// TwinCAT 3 PLC project MC
// ProgramVersion: 3.1.4022.2
// libraries:
//   Tc2_MC2, * (Beckhoff Automation GmbH)
//   Tc2_Standard, * (Beckhoff Automation GmbH)
//   Tc2_System, * (Beckhoff Automation GmbH)
//   Tc3_Module, * (Beckhoff Automation GmbH)
// project tree:
//   DUTs/ Command.TcDUT, Status.TcDUT
//   GVLs/ GVL.TcGVL
//   / PlcTask.TcTTO
//   POUs/ BigArm.TcPOU, Clamp.TcPOU, DrivingWheel1.TcPOU, DrivingWheel2.TcPOU, DrivingWheel3.TcPOU, DrivingWheel4.TcPOU, Flex.TcPOU, MAIN.TcPOU, MiddleArm.TcPOU, Rotation.TcPOU, SmallArm.TcPOU, SwingArm1.TcPOU, SwingArm2.TcPOU, SwingArm3.TcPOU, SwingArm4.TcPOU, Waist.TcPOU
// real-time tasks:
//   TASK PlcTask: cycle T#10ms, priority 20, ADS port 350
//   TASK C++task: cycle T#10ms, priority 1, ADS port 351
// motion (NC):
//   TASK NC-Task 1 SAF: cycle T#2ms, priority 4, ADS port 501
//   TASK NC-Task 1 SVB: cycle T#10ms, priority 8, ADS port 511
//   AXIS DrivingWheel1 (id 1)
//     OtherSettings: AllowMotionCmdToSlave=true
//     encoder EncType=19
//       EncPara: ScaleFactorDenominator=29, Inverse=true, MaxCount=#xffffffff
//     drive DrvType=16
//       DrvPara: Inverse=true, MaxCount=#xffffffff
//         Analog: ScaleFactorActTorque=0.1
//         TimeComp: TaskDelayCycles=1
//     controller CtrType=1
//       CtrPara: PriorControlFactor=1
//         Observer: BandWidth=20
//   AXIS DrivingWheel2 (id 2)
//     OtherSettings: AllowMotionCmdToSlave=true
//     encoder EncType=19
//       EncPara: ScaleFactorDenominator=29, Inverse=true, MaxCount=#xffffffff
//     drive DrvType=16
//       DrvPara: Inverse=true, MaxCount=#xffffffff
//         Analog: ScaleFactorActTorque=0.1
//         TimeComp: TaskDelayCycles=1
//     controller CtrType=1
//       CtrPara: PriorControlFactor=1
//         Observer: BandWidth=20
//   AXIS DrivingWheel3 (id 3)
//     OtherSettings: AllowMotionCmdToSlave=true
//     encoder EncType=19
//       EncPara: ScaleFactorDenominator=29, MaxCount=#xffffffff
//     drive DrvType=16
//       DrvPara: MaxCount=#xffffffff
//         Analog: ScaleFactorActTorque=0.1
//         TimeComp: TaskDelayCycles=1
//     controller CtrType=1
//       CtrPara: PriorControlFactor=1
//         Observer: BandWidth=20
//   AXIS DrivingWheel4 (id 4)
//     OtherSettings: AllowMotionCmdToSlave=true
//     encoder EncType=19
//       EncPara: ScaleFactorDenominator=29, MaxCount=#xffffffff
//     drive DrvType=16
//       DrvPara: MaxCount=#xffffffff
//         Analog: ScaleFactorActTorque=0.1
//         TimeComp: TaskDelayCycles=1
//     controller CtrType=1
//       CtrPara: PriorControlFactor=1
//         Observer: BandWidth=20
//   AXIS SwingArm1 (id 5)
//     OtherSettings: AllowMotionCmdToSlave=true
//     encoder EncType=19
//       EncPara: ScaleFactorDenominator=17.3, MaxCount=#xffffffff
//     drive DrvType=16
//       DrvPara: MaxCount=#xffffffff
//         Analog: ScaleFactorActTorque=0.1
//         TimeComp: TaskDelayCycles=1
//     controller CtrType=1
//       CtrPara: PriorControlFactor=1
//         Observer: BandWidth=20
//   AXIS SwingArm2 (id 6)
//     OtherSettings: AllowMotionCmdToSlave=true
//     encoder EncType=19
//       EncPara: ScaleFactorDenominator=17.3, Inverse=true, MaxCount=#xffffffff
//     drive DrvType=16
//       DrvPara: Inverse=true, MaxCount=#xffffffff
//         Analog: ScaleFactorActTorque=0.1
//         TimeComp: TaskDelayCycles=1
//     controller CtrType=1
//       CtrPara: PriorControlFactor=1
//         Observer: BandWidth=20
//   AXIS SwingArm3 (id 7)
//     OtherSettings: AllowMotionCmdToSlave=true
//     encoder EncType=19
//       EncPara: ScaleFactorDenominator=17.3, MaxCount=#xffffffff
//     drive DrvType=16
//       DrvPara: MaxCount=#xffffffff
//         Analog: ScaleFactorActTorque=0.1
//         TimeComp: TaskDelayCycles=1
//     controller CtrType=1
//       CtrPara: PriorControlFactor=1
//         Observer: BandWidth=20
//   AXIS SwingArm4 (id 8)
//     OtherSettings: AllowMotionCmdToSlave=true
//     encoder EncType=19
//       EncPara: ScaleFactorDenominator=17.3, Inverse=true, MaxCount=#xffffffff
//     drive DrvType=16
//       DrvPara: Inverse=true, MaxCount=#xffffffff
//         Analog: ScaleFactorActTorque=0.1
//         TimeComp: TaskDelayCycles=1
//     controller CtrType=1
//       CtrPara: PriorControlFactor=1
//         Observer: BandWidth=20
//   AXIS Waist (id 9)
//     OtherSettings: AllowMotionCmdToSlave=true
//     encoder EncType=19
//       EncPara: MaxCount=#xffffffff
//     drive DrvType=16
//       DrvPara: MaxCount=#xffffffff
//         Analog: ScaleFactorActTorque=0.1
//         TimeComp: TaskDelayCycles=1
//     controller CtrType=1
//       CtrPara: PriorControlFactor=1
//         Observer: BandWidth=20
//   AXIS BigArm (id 10)
//     General: UnitName=Degree
//     Dynamic: AccelerationMaximum=80, DecelerationMaximum=80, Acceleration=80, Deceleration=80, Jerk=80
//     Velo: RefSearch=10, RefSync=10, SlowManual=10, FastManual=55, Maximum=60
//     OtherSettings: AllowMotionCmdToSlave=true, PulseDistancePos=0.5, PulseDistanceNeg=0.5
//     encoder EncType=19
//       EncPara: ScaleFactorNumerator=0.000686645507813, MaxCount=#xffffffff
//     drive DrvType=16
//       DrvPara: MaxCount=#xffffffff
//         Analog: VeloReferenz=60, ScaleFactorActTorque=0.1
//         TimeComp: TaskDelayCycles=1
//     controller CtrType=1
//       CtrPara: PriorControlFactor=1
//         PID: PosKp=7
//         Observer: BandWidth=20
//   AXIS MiddleArm (id 11)
//     General: UnitName=Degree
//     Dynamic: AccelerationMaximum=80, DecelerationMaximum=80, Acceleration=80, Deceleration=80, Jerk=80
//     Velo: RefSearch=10, RefSync=10, SlowManual=10, FastManual=55, Maximum=60
//     OtherSettings: AllowMotionCmdToSlave=true, PulseDistancePos=0.5, PulseDistanceNeg=0.5
//     encoder EncType=19
//       EncPara: ScaleFactorNumerator=0.000686645507813, MaxCount=#xffffffff
//     drive DrvType=16
//       DrvPara: MaxCount=#xffffffff
//         Analog: VeloReferenz=60, ScaleFactorActTorque=0.1
//         TimeComp: TaskDelayCycles=1
//     controller CtrType=1
//       CtrPara: PriorControlFactor=1
//         PID: PosKp=7
//         Observer: BandWidth=20
//   AXIS SmallArm (id 12)
//     General: UnitName=Degree
//     Dynamic: AccelerationMaximum=80, DecelerationMaximum=80, Acceleration=80, Deceleration=80, Jerk=80
//     Velo: RefSearch=10, RefSync=10, SlowManual=10, FastManual=55, Maximum=60
//     OtherSettings: AllowMotionCmdToSlave=true, PulseDistancePos=0.5, PulseDistanceNeg=0.5
//     encoder EncType=19
//       EncPara: ScaleFactorNumerator=0.000686645507813, Inverse=true, MaxCount=#xffffffff
//     drive DrvType=16
//       DrvPara: Inverse=true, MaxCount=#xffffffff
//         Analog: VeloReferenz=60, ScaleFactorActTorque=0.1
//         TimeComp: TaskDelayCycles=1
//     controller CtrType=1
//       CtrPara: PriorControlFactor=1
//         PID: PosKp=7
//         Observer: BandWidth=20
//   AXIS Rotation (id 13)
//     General: UnitName=Degree
//     Dynamic: AccelerationMaximum=80, DecelerationMaximum=80, Acceleration=80, Deceleration=80, Jerk=80
//     Velo: RefSearch=10, RefSync=10, SlowManual=10, FastManual=55, Maximum=60
//     OtherSettings: AllowMotionCmdToSlave=true, PulseDistancePos=0.5, PulseDistanceNeg=0.5
//     encoder EncType=19
//       EncPara: ScaleFactorNumerator=0.000686645507813, MaxCount=#xffffffff
//     drive DrvType=16
//       DrvPara: MaxCount=#xffffffff
//         Analog: VeloReferenz=60, ScaleFactorActTorque=0.1
//         TimeComp: TaskDelayCycles=1
//     controller CtrType=1
//       CtrPara: PriorControlFactor=1
//         PID: PosKp=7
//         Observer: BandWidth=20
// I/O:
//   DEVICE Device 1 (EtherCAT), AmsNetId 192.168.1.200.2.1
//     Term 1 (EK1200) [EK1200-5000 EtherCAT Power supply (2A E-Bus)]
//       Term 2 (EL6751) [EL6751 CANopen Master]
//       Term 3 (EL9011) [EL9011 End Terminal]
//   DEVICE Device 2 (EL6751), AmsNetId 192.168.1.200.3.1
//     Bigarm
//     MiddleArm
//     SmallArm
//     Rotation
//     Box 1 (Twitter)
//   DEVICE Device 5 (EtherCAT), AmsNetId 192.168.1.200.6.1
//     Drive 8 (Elmo Drive) [Gold EtherCAT GCON Drive Rev:0x00010420]
//     Drive 9 (Elmo Drive) [Gold EtherCAT GCON Drive Rev:0x00010420]
//     Drive 10 (Elmo Drive) [Gold EtherCAT GCON Drive Rev:0x00010420]
//     Drive 11 (Elmo Drive) [Gold EtherCAT GCON Drive Rev:0x00010420]
//     Drive 12 (Elmo Drive) [Gold EtherCAT GCON Drive Rev:0x00010420]
//     Drive 13 (Elmo Drive) [Gold EtherCAT GCON Drive Rev:0x00010420]
//     Drive 14 (Elmo Drive) [Gold EtherCAT GCON Drive Rev:0x00010420]
//     Drive 15 (Elmo Drive) [Gold EtherCAT GCON Drive Rev:0x00010420]
//     Drive 16 (Elmo Drive) [Gold EtherCAT GCON Drive Rev:0x00010420]
// variable links:
//   Device 5 (EtherCAT) <-> LibInterface/LibInterface_Obj1 (LibInterface)
//     Drive 11 (Elmo Drive)/Outputs/Digital Outputs <-> Outputs/lighting
//     Drive 15 (Elmo Drive)/Inputs/Digital Inputs <-> Inputs/jinting
//   NC-Task 1 SAF/Axes/BigArm <-> Device 2 (EL6751)/Bigarm
//     Drive/Inputs/In/nState1 <-> TxPDO 3/Inputs/StatusWord1
//     Drive/Inputs/In/nState2 <-> TxPDO 3/Inputs/StatusWord1 @bit 8
//     Drive/Outputs/Out/nCtrl1 <-> RxPDO 3/Outputs/ControlWord1
//     Drive/Outputs/Out/nCtrl2 <-> RxPDO 3/Outputs/ControlWord1 @bit 8
//     Drive/Outputs/Out/nDataOut1 <-> RxPDO 3/Outputs/TargetPosition1
//     Enc/Inputs/In/nDataIn1 <-> TxPDO 3/Inputs/ActualPosition1
//   NC-Task 1 SAF/Axes/DrivingWheel1 <-> Device 5 (EtherCAT)/Drive 8 (Elmo Drive)
//     Drive/Inputs/In/nDcOutputTime <-> InfoData/DcOutputShift
//     Drive/Inputs/In/nState1 <-> Inputs/Status word
//     Drive/Inputs/In/nState2 <-> Inputs/Status word @bit 8
//     Drive/Inputs/In/nState4 @bit 1 <-> WcState/InputToggle
//     Drive/Inputs/In/nState4 <-> WcState/WcState
//     Drive/Outputs/Out/nCtrl1 <-> Outputs/Control word
//     Drive/Outputs/Out/nCtrl2 <-> Outputs/Control word @bit 8
//     Drive/Outputs/Out/nDataOut1 <-> Outputs/Target Position
//     Enc/Inputs/In/nDataIn1 <-> Inputs/Position actual value
//     Enc/Inputs/In/nDcInputTime <-> InfoData/DcInputShift
//     Enc/Inputs/In/nState4 @bit 1 <-> WcState/InputToggle
//     Enc/Inputs/In/nState4 <-> WcState/WcState
//   NC-Task 1 SAF/Axes/DrivingWheel2 <-> Device 5 (EtherCAT)/Drive 10 (Elmo Drive)
//     Drive/Inputs/In/nDcOutputTime <-> InfoData/DcOutputShift
//     Drive/Inputs/In/nState1 <-> Inputs/Status word
//     Drive/Inputs/In/nState2 <-> Inputs/Status word @bit 8
//     Drive/Inputs/In/nState4 @bit 1 <-> WcState/InputToggle
//     Drive/Inputs/In/nState4 <-> WcState/WcState
//     Drive/Outputs/Out/nCtrl1 <-> Outputs/Control word
//     Drive/Outputs/Out/nCtrl2 <-> Outputs/Control word @bit 8
//     Drive/Outputs/Out/nDataOut1 <-> Outputs/Target Position
//     Enc/Inputs/In/nDataIn1 <-> Inputs/Position actual value
//     Enc/Inputs/In/nDcInputTime <-> InfoData/DcInputShift
//     Enc/Inputs/In/nState4 @bit 1 <-> WcState/InputToggle
//     Enc/Inputs/In/nState4 <-> WcState/WcState
//   NC-Task 1 SAF/Axes/DrivingWheel3 <-> Device 5 (EtherCAT)/Drive 12 (Elmo Drive)
//     Drive/Inputs/In/nDcOutputTime <-> InfoData/DcOutputShift
//     Drive/Inputs/In/nState1 <-> Inputs/Status word
//     Drive/Inputs/In/nState2 <-> Inputs/Status word @bit 8
//     Drive/Inputs/In/nState4 @bit 1 <-> WcState/InputToggle
//     Drive/Inputs/In/nState4 <-> WcState/WcState
//     Drive/Outputs/Out/nCtrl1 <-> Outputs/Control word
//     Drive/Outputs/Out/nCtrl2 <-> Outputs/Control word @bit 8
//     Drive/Outputs/Out/nDataOut1 <-> Outputs/Target Position
//     Enc/Inputs/In/nDataIn1 <-> Inputs/Position actual value
//     Enc/Inputs/In/nDcInputTime <-> InfoData/DcInputShift
//     Enc/Inputs/In/nState4 @bit 1 <-> WcState/InputToggle
//     Enc/Inputs/In/nState4 <-> WcState/WcState
//   NC-Task 1 SAF/Axes/DrivingWheel4 <-> Device 5 (EtherCAT)/Drive 14 (Elmo Drive)
//     Drive/Inputs/In/nDcOutputTime <-> InfoData/DcOutputShift
//     Drive/Inputs/In/nState1 <-> Inputs/Status word
//     Drive/Inputs/In/nState2 <-> Inputs/Status word @bit 8
//     Drive/Inputs/In/nState4 @bit 1 <-> WcState/InputToggle
//     Drive/Inputs/In/nState4 <-> WcState/WcState
//     Drive/Outputs/Out/nCtrl1 <-> Outputs/Control word
//     Drive/Outputs/Out/nCtrl2 <-> Outputs/Control word @bit 8
//     Drive/Outputs/Out/nDataOut1 <-> Outputs/Target Position
//     Enc/Inputs/In/nDataIn1 <-> Inputs/Position actual value
//     Enc/Inputs/In/nDcInputTime <-> InfoData/DcInputShift
//     Enc/Inputs/In/nState4 @bit 1 <-> WcState/InputToggle
//     Enc/Inputs/In/nState4 <-> WcState/WcState
//   NC-Task 1 SAF/Axes/MiddleArm <-> Device 2 (EL6751)/MiddleArm
//     Drive/Inputs/In/nState1 <-> TxPDO 3/Inputs/StatusWord1
//     Drive/Inputs/In/nState2 <-> TxPDO 3/Inputs/StatusWord1 @bit 8
//     Drive/Outputs/Out/nCtrl1 <-> RxPDO 3/Outputs/ControlWord1
//     Drive/Outputs/Out/nCtrl2 <-> RxPDO 3/Outputs/ControlWord1 @bit 8
//     Drive/Outputs/Out/nDataOut1 <-> RxPDO 3/Outputs/TargetPosition1
//     Enc/Inputs/In/nDataIn1 <-> TxPDO 3/Inputs/ActualPosition1
//   NC-Task 1 SAF/Axes/Rotation <-> Device 2 (EL6751)/Rotation
//     Drive/Inputs/In/nState1 <-> TxPDO 3/Inputs/StatusWord1
//     Drive/Inputs/In/nState2 <-> TxPDO 3/Inputs/StatusWord1 @bit 8
//     Drive/Outputs/Out/nCtrl1 <-> RxPDO 3/Outputs/ControlWord1
//     Drive/Outputs/Out/nCtrl2 <-> RxPDO 3/Outputs/ControlWord1 @bit 8
//     Drive/Outputs/Out/nDataOut1 <-> RxPDO 3/Outputs/TargetPosition1
//     Enc/Inputs/In/nDataIn1 <-> TxPDO 3/Inputs/ActualPosition1
//   NC-Task 1 SAF/Axes/SmallArm <-> Device 2 (EL6751)/SmallArm
//     Drive/Inputs/In/nState1 <-> TxPDO 3/Inputs/StatusWord1
//     Drive/Inputs/In/nState2 <-> TxPDO 3/Inputs/StatusWord1 @bit 8
//     Drive/Outputs/Out/nCtrl1 <-> RxPDO 3/Outputs/ControlWord1
//     Drive/Outputs/Out/nCtrl2 <-> RxPDO 3/Outputs/ControlWord1 @bit 8
//     Drive/Outputs/Out/nDataOut1 <-> RxPDO 3/Outputs/TargetPosition1
//     Enc/Inputs/In/nDataIn1 <-> TxPDO 3/Inputs/ActualPosition1
//   NC-Task 1 SAF/Axes/SwingArm1 <-> Device 5 (EtherCAT)/Drive 9 (Elmo Drive)
//     Drive/Inputs/In/nDcOutputTime <-> InfoData/DcOutputShift
//     Drive/Inputs/In/nState1 <-> Inputs/Status word
//     Drive/Inputs/In/nState2 <-> Inputs/Status word @bit 8
//     Drive/Inputs/In/nState4 @bit 1 <-> WcState/InputToggle
//     Drive/Inputs/In/nState4 <-> WcState/WcState
//     Drive/Outputs/Out/nCtrl1 <-> Outputs/Control word
//     Drive/Outputs/Out/nCtrl2 <-> Outputs/Control word @bit 8
//     Drive/Outputs/Out/nDataOut1 <-> Outputs/Target Position
//     Enc/Inputs/In/nDataIn1 <-> Inputs/Position actual value
//     Enc/Inputs/In/nDcInputTime <-> InfoData/DcInputShift
//     Enc/Inputs/In/nState4 @bit 1 <-> WcState/InputToggle
//     Enc/Inputs/In/nState4 <-> WcState/WcState
//   NC-Task 1 SAF/Axes/SwingArm2 <-> Device 5 (EtherCAT)/Drive 11 (Elmo Drive)
//     Drive/Inputs/In/nDcOutputTime <-> InfoData/DcOutputShift
//     Drive/Inputs/In/nState1 <-> Inputs/Status word
//     Drive/Inputs/In/nState2 <-> Inputs/Status word @bit 8
//     Drive/Inputs/In/nState4 @bit 1 <-> WcState/InputToggle
//     Drive/Inputs/In/nState4 <-> WcState/WcState
//     Drive/Outputs/Out/nCtrl1 <-> Outputs/Control word
//     Drive/Outputs/Out/nCtrl2 <-> Outputs/Control word @bit 8
//     Drive/Outputs/Out/nDataOut1 <-> Outputs/Target Position
//     Enc/Inputs/In/nDataIn1 <-> Inputs/Position actual value
//     Enc/Inputs/In/nDcInputTime <-> InfoData/DcInputShift
//     Enc/Inputs/In/nState4 @bit 1 <-> WcState/InputToggle
//     Enc/Inputs/In/nState4 <-> WcState/WcState
//   NC-Task 1 SAF/Axes/SwingArm3 <-> Device 5 (EtherCAT)/Drive 13 (Elmo Drive)
//     Drive/Inputs/In/nDcOutputTime <-> InfoData/DcOutputShift
//     Drive/Inputs/In/nState1 <-> Inputs/Status word
//     Drive/Inputs/In/nState2 <-> Inputs/Status word @bit 8
//     Drive/Inputs/In/nState4 @bit 1 <-> WcState/InputToggle
//     Drive/Inputs/In/nState4 <-> WcState/WcState
//     Drive/Outputs/Out/nCtrl1 <-> Outputs/Control word
//     Drive/Outputs/Out/nCtrl2 <-> Outputs/Control word @bit 8
//     Drive/Outputs/Out/nDataOut1 <-> Outputs/Target Position
//     Enc/Inputs/In/nDataIn1 <-> Inputs/Position actual value
//     Enc/Inputs/In/nDcInputTime <-> InfoData/DcInputShift
//     Enc/Inputs/In/nState4 @bit 1 <-> WcState/InputToggle
//     Enc/Inputs/In/nState4 <-> WcState/WcState
//   NC-Task 1 SAF/Axes/SwingArm4 <-> Device 5 (EtherCAT)/Drive 15 (Elmo Drive)
//     Drive/Inputs/In/nDcOutputTime <-> InfoData/DcOutputShift
//     Drive/Inputs/In/nState1 <-> Inputs/Status word
//     Drive/Inputs/In/nState2 <-> Inputs/Status word @bit 8
//     Drive/Inputs/In/nState4 @bit 1 <-> WcState/InputToggle
//     Drive/Inputs/In/nState4 <-> WcState/WcState
//     Drive/Outputs/Out/nCtrl1 <-> Outputs/Control word
//     Drive/Outputs/Out/nCtrl2 <-> Outputs/Control word @bit 8
//     Drive/Outputs/Out/nDataOut1 <-> Outputs/Target Position
//     Enc/Inputs/In/nDataIn1 <-> Inputs/Position actual value
//     Enc/Inputs/In/nDcInputTime <-> InfoData/DcInputShift
//     Enc/Inputs/In/nState4 @bit 1 <-> WcState/InputToggle
//     Enc/Inputs/In/nState4 <-> WcState/WcState
//   NC-Task 1 SAF/Axes/Waist <-> Device 5 (EtherCAT)/Drive 16 (Elmo Drive)
//     Drive/Inputs/In/nDcOutputTime <-> InfoData/DcOutputShift
//     Drive/Inputs/In/nState1 <-> Inputs/Status word
//     Drive/Inputs/In/nState2 <-> Inputs/Status word @bit 8
//     Drive/Inputs/In/nState4 @bit 1 <-> WcState/InputToggle
//     Drive/Inputs/In/nState4 <-> WcState/WcState
//     Drive/Outputs/Out/nCtrl1 <-> Outputs/Control word
//     Drive/Outputs/Out/nCtrl2 <-> Outputs/Control word @bit 8
//     Drive/Outputs/Out/nDataOut1 <-> Outputs/Target Position
//     Enc/Inputs/In/nDataIn1 <-> Inputs/Position actual value
//     Enc/Inputs/In/nDcInputTime <-> InfoData/DcInputShift
//     Enc/Inputs/In/nState4 @bit 1 <-> WcState/InputToggle
//     Enc/Inputs/In/nState4 <-> WcState/WcState
//   MC/MC Instance <-> Device 2 (EL6751)/Box 1 (Twitter)
//     PlcTask Inputs/GVL.Astatusword[1] <-> TxPDO 1/Inputs/statusword
//     PlcTask Inputs/GVL.readActualpostion[1] <-> TxPDO 1/Inputs/Actualpostion
//     PlcTask Inputs/GVL.readIOStatus[1] <-> TxPDO 2/Inputs/DI
//     PlcTask Outputs/GVL.Acontrolword[1] <-> RxPDO 1/Outputs/Controlword
//     PlcTask Outputs/GVL.SetActualVelocity[1] <-> RxPDO 2/Outputs/TargetVelocity
//     PlcTask Outputs/GVL.SetUnitmode[1] <-> RxPDO 2/Outputs/unitmode
//   MC/MC Instance <-> NC-Task 1 SAF/Axes/BigArm
//     PlcTask Inputs/MAIN.fbBigArm.axis.NcToPlc <-> Outputs/ToPlc
//     PlcTask Outputs/MAIN.fbBigArm.axis.PlcToNc <-> Inputs/FromPlc
//   MC/MC Instance <-> NC-Task 1 SAF/Axes/DrivingWheel1
//     PlcTask Inputs/MAIN.fbDrivingWheel1.axis.NcToPlc <-> Outputs/ToPlc
//     PlcTask Outputs/MAIN.fbDrivingWheel1.axis.PlcToNc <-> Inputs/FromPlc
//   MC/MC Instance <-> NC-Task 1 SAF/Axes/DrivingWheel2
//     PlcTask Inputs/MAIN.fbDrivingWheel2.axis.NcToPlc <-> Outputs/ToPlc
//     PlcTask Outputs/MAIN.fbDrivingWheel2.axis.PlcToNc <-> Inputs/FromPlc
//   MC/MC Instance <-> NC-Task 1 SAF/Axes/DrivingWheel3
//     PlcTask Inputs/MAIN.fbDrivingWheel3.axis.NcToPlc <-> Outputs/ToPlc
//     PlcTask Outputs/MAIN.fbDrivingWheel3.axis.PlcToNc <-> Inputs/FromPlc
//   MC/MC Instance <-> NC-Task 1 SAF/Axes/DrivingWheel4
//     PlcTask Inputs/MAIN.fbDrivingWheel4.axis.NcToPlc <-> Outputs/ToPlc
//     PlcTask Outputs/MAIN.fbDrivingWheel4.axis.PlcToNc <-> Inputs/FromPlc
//   MC/MC Instance <-> NC-Task 1 SAF/Axes/MiddleArm
//     PlcTask Inputs/MAIN.fbMiddleArm.axis.NcToPlc <-> Outputs/ToPlc
//     PlcTask Outputs/MAIN.fbMiddleArm.axis.PlcToNc <-> Inputs/FromPlc
//   MC/MC Instance <-> NC-Task 1 SAF/Axes/Rotation
//     PlcTask Inputs/MAIN.fbRotation.axis.NcToPlc <-> Outputs/ToPlc
//     PlcTask Outputs/MAIN.fbRotation.axis.PlcToNc <-> Inputs/FromPlc
//   MC/MC Instance <-> NC-Task 1 SAF/Axes/SmallArm
//     PlcTask Inputs/MAIN.fbSmallArm.axis.NcToPlc <-> Outputs/ToPlc
//     PlcTask Outputs/MAIN.fbSmallArm.axis.PlcToNc <-> Inputs/FromPlc
//   MC/MC Instance <-> NC-Task 1 SAF/Axes/SwingArm1
//     PlcTask Inputs/MAIN.fbSwingArm1.axis.NcToPlc <-> Outputs/ToPlc
//     PlcTask Outputs/MAIN.fbSwingArm1.axis.PlcToNc <-> Inputs/FromPlc
//   MC/MC Instance <-> NC-Task 1 SAF/Axes/SwingArm2
//     PlcTask Inputs/MAIN.fbSwingArm2.axis.NcToPlc <-> Outputs/ToPlc
//     PlcTask Outputs/MAIN.fbSwingArm2.axis.PlcToNc <-> Inputs/FromPlc
//   MC/MC Instance <-> NC-Task 1 SAF/Axes/SwingArm3
//     PlcTask Inputs/MAIN.fbSwingArm3.axis.NcToPlc <-> Outputs/ToPlc
//     PlcTask Outputs/MAIN.fbSwingArm3.axis.PlcToNc <-> Inputs/FromPlc
//   MC/MC Instance <-> NC-Task 1 SAF/Axes/SwingArm4
//     PlcTask Inputs/MAIN.fbSwingArm4.axis.NcToPlc <-> Outputs/ToPlc
//     PlcTask Outputs/MAIN.fbSwingArm4.axis.PlcToNc <-> Inputs/FromPlc
//   MC/MC Instance <-> NC-Task 1 SAF/Axes/Waist
//     PlcTask Inputs/MAIN.fbWaist.axis.NcToPlc <-> Outputs/ToPlc
//     PlcTask Outputs/MAIN.fbWaist.axis.PlcToNc <-> Inputs/FromPlc
//   MC/MC Instance <-> LibInterface/LibInterface_Obj1 (LibInterface)
//     PlcTask Inputs/MAIN.BigArmInput/Enable <-> Outputs/BigArmInput/Enable
//     PlcTask Inputs/MAIN.BigArmInput/Halt <-> Outputs/BigArmInput/Halt
//     PlcTask Inputs/MAIN.BigArmInput/Home <-> Outputs/BigArmInput/Home
//     PlcTask Inputs/MAIN.BigArmInput/Move_Absolute <-> Outputs/BigArmInput/MoveAbsolute
//     PlcTask Inputs/MAIN.BigArmInput/Move_Relative <-> Outputs/BigArmInput/MoveRelative
//     PlcTask Inputs/MAIN.BigArmInput/Move_Velocity <-> Outputs/BigArmInput/MoveVelocity
//     PlcTask Inputs/MAIN.BigArmInput/Position <-> Outputs/BigArmInput/Position
//     PlcTask Inputs/MAIN.BigArmInput/Reset <-> Outputs/BigArmInput/Reset
//     PlcTask Inputs/MAIN.BigArmInput/SetZero <-> Outputs/BigArmInput/SetZero
//     PlcTask Inputs/MAIN.BigArmInput/Velocity <-> Outputs/BigArmInput/Velocity
//     PlcTask Inputs/MAIN.DrivingWheel{1..4}Input/Enable <-> Outputs/DrivingWheel{1..4}Input/Enable  (4 links)
//     PlcTask Inputs/MAIN.DrivingWheel{1..4}Input/Halt <-> Outputs/DrivingWheel{1..4}Input/Halt  (4 links)
//     PlcTask Inputs/MAIN.DrivingWheel{1..4}Input/Home <-> Outputs/DrivingWheel{1..4}Input/Home  (4 links)
//     PlcTask Inputs/MAIN.DrivingWheel{1..4}Input/Move_Absolute <-> Outputs/DrivingWheel{1..4}Input/MoveAbsolute  (4 links)
//     PlcTask Inputs/MAIN.DrivingWheel{1..4}Input/Move_Relative <-> Outputs/DrivingWheel{1..4}Input/MoveRelative  (4 links)
//     PlcTask Inputs/MAIN.DrivingWheel{1..4}Input/Move_Velocity <-> Outputs/DrivingWheel{1..4}Input/MoveVelocity  (4 links)
//     PlcTask Inputs/MAIN.DrivingWheel{1..4}Input/Position <-> Outputs/DrivingWheel{1..4}Input/Position  (4 links)
//     PlcTask Inputs/MAIN.DrivingWheel{1..4}Input/Reset <-> Outputs/DrivingWheel{1..4}Input/Reset  (4 links)
//     PlcTask Inputs/MAIN.DrivingWheel{1..4}Input/SetZero <-> Outputs/DrivingWheel{1..4}Input/SetZero  (4 links)
//     PlcTask Inputs/MAIN.DrivingWheel{1..4}Input/Velocity <-> Outputs/DrivingWheel{1..4}Input/Velocity  (4 links)
//     PlcTask Inputs/MAIN.FlexInput/Enable <-> Outputs/FlexInput/Enable
//     PlcTask Inputs/MAIN.FlexInput/Halt <-> Outputs/FlexInput/Halt
//     PlcTask Inputs/MAIN.FlexInput/Home <-> Outputs/FlexInput/Home
//     PlcTask Inputs/MAIN.FlexInput/Move_Absolute <-> Outputs/FlexInput/MoveAbsolute
//     PlcTask Inputs/MAIN.FlexInput/Move_Relative <-> Outputs/FlexInput/MoveRelative
//     PlcTask Inputs/MAIN.FlexInput/Move_Velocity <-> Outputs/FlexInput/MoveVelocity
//     PlcTask Inputs/MAIN.FlexInput/Position <-> Outputs/FlexInput/Position
//     PlcTask Inputs/MAIN.FlexInput/Reset <-> Outputs/FlexInput/Reset
//     PlcTask Inputs/MAIN.FlexInput/SetZero <-> Outputs/FlexInput/SetZero
//     PlcTask Inputs/MAIN.FlexInput/Velocity <-> Outputs/FlexInput/Velocity
//     PlcTask Inputs/MAIN.GripperEnable <-> Outputs/ClampInput/Enable
//     PlcTask Inputs/MAIN.GripperSetSpeed <-> Outputs/ClampInput/SetSpped
//     PlcTask Inputs/MAIN.MiddleArmInput/Enable <-> Outputs/MiddleArmInput/Enable
//     PlcTask Inputs/MAIN.MiddleArmInput/Halt <-> Outputs/MiddleArmInput/Halt
//     PlcTask Inputs/MAIN.MiddleArmInput/Home <-> Outputs/MiddleArmInput/Home
//     PlcTask Inputs/MAIN.MiddleArmInput/Move_Absolute <-> Outputs/MiddleArmInput/MoveAbsolute
//     PlcTask Inputs/MAIN.MiddleArmInput/Move_Relative <-> Outputs/MiddleArmInput/MoveRelative
//     PlcTask Inputs/MAIN.MiddleArmInput/Move_Velocity <-> Outputs/MiddleArmInput/MoveVelocity
//     PlcTask Inputs/MAIN.MiddleArmInput/Position <-> Outputs/MiddleArmInput/Position
//     PlcTask Inputs/MAIN.MiddleArmInput/Reset <-> Outputs/MiddleArmInput/Reset
//     PlcTask Inputs/MAIN.MiddleArmInput/SetZero <-> Outputs/MiddleArmInput/SetZero
//     PlcTask Inputs/MAIN.MiddleArmInput/Velocity <-> Outputs/MiddleArmInput/Velocity
//     PlcTask Inputs/MAIN.RotationInput/Enable <-> Outputs/RotationInput/Enable
//     PlcTask Inputs/MAIN.RotationInput/Halt <-> Outputs/RotationInput/Halt
//     PlcTask Inputs/MAIN.RotationInput/Home <-> Outputs/RotationInput/Home
//     PlcTask Inputs/MAIN.RotationInput/Move_Absolute <-> Outputs/RotationInput/MoveAbsolute
//     PlcTask Inputs/MAIN.RotationInput/Move_Relative <-> Outputs/RotationInput/MoveRelative
//     PlcTask Inputs/MAIN.RotationInput/Move_Velocity <-> Outputs/RotationInput/MoveVelocity
//     PlcTask Inputs/MAIN.RotationInput/Position <-> Outputs/RotationInput/Position
//     PlcTask Inputs/MAIN.RotationInput/Reset <-> Outputs/RotationInput/Reset
//     PlcTask Inputs/MAIN.RotationInput/SetZero <-> Outputs/RotationInput/SetZero
//     PlcTask Inputs/MAIN.RotationInput/Velocity <-> Outputs/RotationInput/Velocity
//     PlcTask Inputs/MAIN.SmallArmInput/Enable <-> Outputs/SmallArmInput/Enable
//     PlcTask Inputs/MAIN.SmallArmInput/Halt <-> Outputs/SmallArmInput/Halt
//     PlcTask Inputs/MAIN.SmallArmInput/Home <-> Outputs/SmallArmInput/Home
//     PlcTask Inputs/MAIN.SmallArmInput/Move_Absolute <-> Outputs/SmallArmInput/MoveAbsolute
//     PlcTask Inputs/MAIN.SmallArmInput/Move_Relative <-> Outputs/SmallArmInput/MoveRelative
//     PlcTask Inputs/MAIN.SmallArmInput/Move_Velocity <-> Outputs/SmallArmInput/MoveVelocity
//     PlcTask Inputs/MAIN.SmallArmInput/Position <-> Outputs/SmallArmInput/Position
//     PlcTask Inputs/MAIN.SmallArmInput/Reset <-> Outputs/SmallArmInput/Reset
//     PlcTask Inputs/MAIN.SmallArmInput/SetZero <-> Outputs/SmallArmInput/SetZero
//     PlcTask Inputs/MAIN.SmallArmInput/Velocity <-> Outputs/SmallArmInput/Velocity
//     PlcTask Inputs/MAIN.SwingArm{1..4}Input/Enable <-> Outputs/SwingArm{1..4}Input/Enable  (4 links)
//     PlcTask Inputs/MAIN.SwingArm{1..4}Input/Halt <-> Outputs/SwingArm{1..4}Input/Halt  (4 links)
//     PlcTask Inputs/MAIN.SwingArm{1..4}Input/Home <-> Outputs/SwingArm{1..4}Input/Home  (4 links)
//     PlcTask Inputs/MAIN.SwingArm{1..4}Input/Move_Absolute <-> Outputs/SwingArm{1..4}Input/MoveAbsolute  (4 links)
//     PlcTask Inputs/MAIN.SwingArm{1..4}Input/Move_Relative <-> Outputs/SwingArm{1..4}Input/MoveRelative  (4 links)
//     PlcTask Inputs/MAIN.SwingArm{1..4}Input/Move_Velocity <-> Outputs/SwingArm{1..4}Input/MoveVelocity  (4 links)
//     PlcTask Inputs/MAIN.SwingArm{1..4}Input/Position <-> Outputs/SwingArm{1..4}Input/Position  (4 links)
//     PlcTask Inputs/MAIN.SwingArm{1..4}Input/Reset <-> Outputs/SwingArm{1..4}Input/Reset  (4 links)
//     PlcTask Inputs/MAIN.SwingArm{1..4}Input/SetZero <-> Outputs/SwingArm{1..4}Input/SetZero  (4 links)
//     PlcTask Inputs/MAIN.SwingArm{1..4}Input/Velocity <-> Outputs/SwingArm{1..4}Input/Velocity  (4 links)
//     PlcTask Inputs/MAIN.WaistInput/Enable <-> Outputs/WaistInput/Enable
//     PlcTask Inputs/MAIN.WaistInput/Halt <-> Outputs/WaistInput/Halt
//     PlcTask Inputs/MAIN.WaistInput/Home <-> Outputs/WaistInput/Home
//     PlcTask Inputs/MAIN.WaistInput/Move_Absolute <-> Outputs/WaistInput/MoveAbsolute
//     PlcTask Inputs/MAIN.WaistInput/Move_Relative <-> Outputs/WaistInput/MoveRelative
//     PlcTask Inputs/MAIN.WaistInput/Move_Velocity <-> Outputs/WaistInput/MoveVelocity
//     PlcTask Inputs/MAIN.WaistInput/Position <-> Outputs/WaistInput/Position
//     PlcTask Inputs/MAIN.WaistInput/Reset <-> Outputs/WaistInput/Reset
//     PlcTask Inputs/MAIN.WaistInput/SetZero <-> Outputs/WaistInput/SetZero
//     PlcTask Inputs/MAIN.WaistInput/Velocity <-> Outputs/WaistInput/Velocity
//     PlcTask Outputs/MAIN.BigArmOutput/Enable <-> Inputs/BigArmOutput/Enable
//     PlcTask Outputs/MAIN.BigArmOutput/Position <-> Inputs/BigArmOutput/Position
//     PlcTask Outputs/MAIN.BigArmOutput/Velocity <-> Inputs/BigArmOutput/Velocity
//     PlcTask Outputs/MAIN.DrivingWheel{1..4}Output/Enable <-> Inputs/DrivingWheel{1..4}Output/Enable  (4 links)
//     PlcTask Outputs/MAIN.DrivingWheel{1..4}Output/Position <-> Inputs/DrivingWheel{1..4}Output/Position  (4 links)
//     PlcTask Outputs/MAIN.DrivingWheel{1..4}Output/Velocity <-> Inputs/DrivingWheel{1..4}Output/Velocity  (4 links)
//     PlcTask Outputs/MAIN.FlexOutput/Enable <-> Inputs/FlexOutput/Enable
//     PlcTask Outputs/MAIN.FlexOutput/Position <-> Inputs/FlexOutput/Position
//     PlcTask Outputs/MAIN.FlexOutput/Velocity <-> Inputs/FlexOutput/Velocity
//     PlcTask Outputs/MAIN.GripperIOStatus <-> Inputs/ClampOutput/IO
//     PlcTask Outputs/MAIN.GripperReadPos <-> Inputs/ClampOutput/Position
//     PlcTask Outputs/MAIN.MiddleArmOutput/Enable <-> Inputs/MiddleArmOutput/Enable
//     PlcTask Outputs/MAIN.MiddleArmOutput/Position <-> Inputs/MiddleArmOutput/Position
//     PlcTask Outputs/MAIN.MiddleArmOutput/Velocity <-> Inputs/MiddleArmOutput/Velocity
//     PlcTask Outputs/MAIN.RotationOutput/Enable <-> Inputs/RotationOutput/Enable
//     PlcTask Outputs/MAIN.RotationOutput/Position <-> Inputs/RotationOutput/Position
//     PlcTask Outputs/MAIN.RotationOutput/Velocity <-> Inputs/RotationOutput/Velocity
//     PlcTask Outputs/MAIN.SmallArmOutput/Enable <-> Inputs/SmallArmOutput/Enable
//     PlcTask Outputs/MAIN.SmallArmOutput/Position <-> Inputs/SmallArmOutput/Position
//     PlcTask Outputs/MAIN.SmallArmOutput/Velocity <-> Inputs/SmallArmOutput/Velocity
//     PlcTask Outputs/MAIN.SwingArm{1..4}Output/Enable <-> Inputs/SwingArm{1..4}Output/Enable  (4 links)
//     PlcTask Outputs/MAIN.SwingArm{1..4}Output/Position <-> Inputs/SwingArm{1..4}Output/Position  (4 links)
//     PlcTask Outputs/MAIN.SwingArm{1..4}Output/Velocity <-> Inputs/SwingArm{1..4}Output/Velocity  (4 links)
//     PlcTask Outputs/MAIN.WaistOutput/Enable <-> Inputs/WaistOutput/Enable
//     PlcTask Outputs/MAIN.WaistOutput/Position <-> Inputs/WaistOutput/Position
//     PlcTask Outputs/MAIN.WaistOutput/Velocity <-> Inputs/WaistOutput/Velocity

CONFIGURATION MC
    RESOURCE PLC ON TwinCAT3
        TASK PlcTask(INTERVAL := T#10ms, PRIORITY := 20);
        PROGRAM MAIN WITH PlcTask : MAIN;
    END_RESOURCE
END_CONFIGURATION

// ---- DUTs/Command.TcDUT
TYPE Command :
STRUCT
	Enable:BOOL;					//使能触发位
	Move_Absolute:BOOL;				//绝对运动触发位
	Move_Relative:BOOL;				//相对运动触发位
	Move_Velocity:BOOL;				//匀速运动触发位
	Reset:BOOL;						//复位触发位
	Halt:BOOL;						//暂停触发位
	Home:BOOL;						//暂停触发位
	SetZero:BOOL;					//设置位置触发位
	Velocity:LREAL;					//速度变量
	Position:LREAL;					//位置变量
	HomeSignal:DINT;				//寻参触发点
END_STRUCT
END_TYPE

// ---- DUTs/Status.TcDUT
TYPE Status :
STRUCT
	Enable:BOOL;					//使能状态
	Velocity:LREAL;					//速度状态
	Position:LREAL;					//位置状态
END_STRUCT
END_TYPE

// ---- GVLs/GVL.TcGVL
{attribute 'qualified_only'}
VAR_GLOBAL
	Acontrolword  AT%Q*:ARRAY[1..1]OF UINT;
	
	SetActualVelocity AT%Q*:ARRAY[1..1]OF DINT;
	SetUnitmode AT%Q*:ARRAY[1..1]OF BYTE;
	
	
	
	Astatusword AT%I*:ARRAY[1..1]OF UINT;
	readActualpostion AT%I*:ARRAY[1..1]OF DINT;
	readActualCurrent AT%I*:ARRAY[1..1]OF UINT;
	readIOStatus AT%I*:ARRAY[1..1]OF DINT;
	
	bigarm_position:LREAL;
	middlearm_position:LREAL;
	
	
	
END_VAR

// ---- POUs/MAIN.TcPOU
PROGRAM MAIN
VAR
	fbDrivingWheel1:DrivingWheel1;				//调用控制驱动轮1功能块
	fbDrivingWheel2:DrivingWheel2;				//调用控制驱动轮2功能块
	fbDrivingWheel3:DrivingWheel3;				//调用控制驱动轮3功能块
	fbDrivingWheel4:DrivingWheel4;				//调用控制驱动轮4功能块
	fbSwingArm1:SwingArm1;						//调用控制摆臂1功能块
	fbSwingArm2:SwingArm2;						//调用控制摆臂2功能块
	fbSwingArm3:SwingArm3;						//调用控制摆臂3功能块
	fbSwingArm4:SwingArm4;						//调用控制摆臂4功能块
	fbWaist:Waist;								//调用控制腰功能块
	fbBigArm:BigArm;							//调用控制大臂功能块
	fbFlex:Flex;								//调用控制伸缩功能块
	fbMiddleArm:MiddleArm;						//调用控制中臂功能块
	fbSmallArm:SmallArm;						//调用控制小臂功能块
	fbRotation:Rotation;						//调用控制旋转功能块
	fbClamp:Clamp;								//调用控制夹紧功能块
//***************************************************************//
	DrivingWheel1Input AT%I*:Command;//驱动轮1PLC轴输入变量
	DrivingWheel2Input AT%I*:Command;//驱动轮2PLC轴输入变量
	DrivingWheel3Input AT%I*:Command;//驱动轮3PLC轴输入变量
	DrivingWheel4Input AT%I*:Command;//驱动轮4PLC轴输入变量
	SwingArm1Input AT%I*:Command;	 //摆臂1PLC轴输入变量
	SwingArm2Input AT%I*:Command;	 //摆臂2PLC轴输入变量
	SwingArm3Input AT%I*:Command;	 //摆臂3PLC轴输入变量
	SwingArm4Input AT%I*:Command;	 //摆臂4PLC轴输入变量
	WaistInput AT%I*:Command;	 	 //腰PLC轴输入变量
	BigArmInput AT%I*:Command;		 //大臂PLC轴输入变量
	FlexInput AT%I*:Command;		 //伸缩PLC轴输入变量
	MiddleArmInput AT%I*:Command;	 //中臂PLC轴输入变量
	SmallArmInput AT%I*:Command;	 //小臂PLC轴输入变量
	RotationInput AT%I*:Command;	 //旋转PLC轴输入变量
	ClampInput AT%I*:Command;		 //夹紧PLC轴输入变量
//***************************************************************//
	DrivingWheel1Output AT%Q*:Status;//驱动轮1PLC轴输出变量
	DrivingWheel2Output AT%Q*:Status;//驱动轮2PLC轴输出变量
	DrivingWheel3Output AT%Q*:Status;//驱动轮3LC轴输出变量
	DrivingWheel4Output AT%Q*:Status;//驱动轮4PLC轴输出变量
	SwingArm1Output AT%Q*:Status;//摆臂1PLC轴输出变量
	SwingArm2Output AT%Q*:Status;//摆臂2PLC轴输出变量
	SwingArm3Output AT%Q*:Status;//摆臂3PLC轴输出变量
	SwingArm4Output AT%Q*:Status;//摆臂4PLC轴输出变量
	WaistOutput AT%Q*:Status; //腰PLC轴输出变量
	BigArmOutput AT%Q*:Status;//大臂PLC轴输出变量
	FlexOutput AT%Q*:Status; //伸缩PLC轴输出变量
	MiddleArmOutput AT%Q*:Status;//中臂PLC轴输出变量
	SmallArmOutput AT%Q*:Status;//小臂PLC轴输出变量
	RotationOutput AT%Q*:Status;//旋转PLC轴输出变量
	ClampOutput AT%Q*:Status;//夹紧PLC轴输出变量
	///////////////////////////////////////////////////////
	GripperEnable AT%I*:DINT;
	GripperSetSpeed AT%I*:DINT;
	GripperReadPos AT%Q*:DINT;
	GripperIOStatus AT%Q*:DINT;
END_VAR


fbDrivingWheel1( AxisInput:=DrivingWheel1Input , AxisOutput=>DrivingWheel1Output );
fbDrivingWheel2( AxisInput:=DrivingWheel2Input , AxisOutput=>DrivingWheel2Output );
fbDrivingWheel3( AxisInput:=DrivingWheel3Input , AxisOutput=>DrivingWheel3Output );
fbDrivingWheel4( AxisInput:=DrivingWheel4Input , AxisOutput=>DrivingWheel4Output );

fbSwingArm1( AxisInput:=SwingArm1Input , AxisOutput=>SwingArm1Output );
fbSwingArm2( AxisInput:=SwingArm2Input , AxisOutput=>SwingArm2Output );
fbSwingArm3( AxisInput:=SwingArm3Input , AxisOutput=>SwingArm3Output );
fbSwingArm4( AxisInput:=SwingArm4Input , AxisOutput=>SwingArm4Output );

fbWaist( AxisInput:=WaistInput , AxisOutput=>WaistOutput );
fbBigArm( AxisInput:=BigArmInput , AxisOutput=>BigArmOutput );
fbFlex(AxisInput:=FlexInput, AxisOutput=>FlexOutput);
fbMiddleArm( AxisInput:=MiddleArmInput , AxisOutput=>MiddleArmOutput );
fbSmallArm( AxisInput:=SmallArmInput , AxisOutput=>SmallArmOutput );
fbRotation( AxisInput:=RotationInput , AxisOutput=>RotationOutput );
fbClamp( AxisInput:=ClampInput , AxisOutput=>ClampOutput );

//////////////////////////////////////////////////////////////////////
//Enable
//when receive enable signal,then gripper driver would be enabled in 3 circles
IF(GripperEnable=1 AND NOT(GVL.Acontrolword[1] =15))THEN
	IF(NOT(GVL.Acontrolword[1] =6) AND NOT(GVL.Acontrolword[1] =7))THEN
			GVL.Acontrolword[1] :=6;		
	ELSIF(GVL.Acontrolword[1] =6)THEN
			GVL.Acontrolword[1] :=7;	
	ELSE
			GVL.Acontrolword[1] :=15;	
			//set driver mode
			GVL.SetUnitmode[1]:=3;
	END_IF
END_IF

//disable
//when receive disnable signal,then gripper driver would be disnabled immediately
IF(GripperEnable=0)THEN
	GVL.Acontrolword[1] :=0;	
END_IF


//set gripper speed,positive speed represent open ,negative speed represent close
IF(GripperEnable=1)THEN
	IF(GripperSetSpeed>100)THEN
		GVL.SetActualVelocity[1]:=100*1000;
	ELSIF(GripperSetSpeed<-100)THEN
		GVL.SetActualVelocity[1]:=-100*1000;
	END_IF
	GVL.SetActualVelocity[1]:=GripperSetSpeed*1000;
END_IF
GripperReadPos:=GVL.readActualpostion[1];
//18bit is the postion-constraint switch
GripperIOStatus:=GVL.readIOStatus[1];

END_PROGRAM

// ---- POUs/DrivingWheel1.TcPOU
FUNCTION_BLOCK DrivingWheel1
VAR_INPUT
	AxisInput:Command;//定义一个驱动轮PLC轴的输入结构体变量
END_VAR
VAR_OUTPUT
	AxisOutput:Status;//定义一个驱动轮PLC轴的输出结构体变量
END_VAR
VAR
	axis:axis_ref;		//定义一个轴
	power:mc_power;		//使能功能块
	moveAbsolute:mc_moveabsolute;//绝对运动功能块
	moveRelative:mc_moverelative;//相对运动功能块
	moveVelocity:mc_movevelocity;//匀速运动功能块
	reset:mc_reset;				//复位功能块
	halt:mc_halt;				//暂停功能块
	Home:mc_home;				//寻参功能块
	SetZero:mc_Setposition;		//强制设置位置功能块
	Dir: MC_Direction;			//匀速运动方向变量，1/3
	Signal:BOOL;				//寻参触发点
END_VAR

power(
	Axis:=axis, 
	Enable:=AxisInput.Enable, 
	Enable_Positive:=TRUE, 
	Enable_Negative:=TRUE, 
	Override:= , 
	BufferMode:= , 
	Options:= , 
	Status=>AxisOutput.Enable, 
	Busy=> , 
	Active=> , 
	Error=> , 
	ErrorID=> );
	
moveAbsolute(
	Axis:=axis, 
	Execute:=AxisInput.Move_Absolute, 
	Position:=AxisInput.Position, 
	Velocity:=AxisInput.Velocity, 
	Acceleration:= , 
	Deceleration:= , 
	Jerk:= , 
	BufferMode:= , 
	Options:= , 
	Done=> , 
	Busy=> , 
	Active=> , 
	CommandAborted=> , 
	Error=> , 
	ErrorID=> );

moveRelative(
	Axis:=axis, 
	Execute:=AxisInput.Move_Relative, 
	Distance:=AxisInput.Position, 
	Velocity:=AxisInput.Velocity, 
	Acceleration:= , 
	Deceleration:= , 
	Jerk:= , 
	BufferMode:= , 
	Options:= , 
	Done=> , 
	Busy=> , 
	Active=> , 
	CommandAborted=> , 
	Error=> , 
	ErrorID=> );

	IF(AxisInput.Velocity>=0)THEN
		Dir:=1;
	ELSIF(AxisInput.Velocity<0)THEN
		Dir:=3;
		AxisInput.Velocity:=-AxisInput.Velocity;
	END_IF
moveVelocity(
	Axis:= axis, 
	Execute:= AxisInput.Move_Velocity, 
	Velocity:= AxisInput.Velocity, 
	Acceleration:= , 
	Deceleration:= , 
	Jerk:= , 
	Direction:= Dir, 
	BufferMode:= , 
	Options:= , 
	InVelocity=> , 
	Busy=> , 
	Active=> , 
	CommandAborted=> , 
	Error=> , 
	ErrorID=> );
	
reset(
	Axis:= axis, 
	Execute:= AxisInput.Reset, 
	Done=> , 
	Busy=> , 
	Error=> , 
	ErrorID=> );
	
halt(
	Axis:= axis, 
	Execute:= AxisInput.Halt, 
	Deceleration:= , 
	Jerk:= , 
	BufferMode:= , 
	Options:= , 
	Done=> , 
	Busy=> , 
	Active=> , 
	CommandAborted=> , 
	Error=> , 
	ErrorID=> );
	IF(AxisInput.HomeSignal=524288)THEN
		Signal:=TRUE;
	ELSE 
		Signal:=FALSE;		
	END_IF	
Home(
	Axis:= axis, 
	Execute:= AxisInput.Home, 
	Position:= 0, 
	HomingMode:= , 
	BufferMode:= , 
	Options:= , 
	bCalibrationCam:= Signal, 
	Done=> , 
	Busy=> , 
	Active=> , 
	CommandAborted=> , 
	Error=> , 
	ErrorID=> );
	
SetZero(
	Axis:=axis , 
	Execute:=AxisInput.SetZero , 
	Position:= 0, 
	Mode:= , 
	Options:= , 
	Done=> , 
	Busy=> , 
	Error=> , 
	ErrorID=> );
AxisOutput.Position:=Axis.NcToPlc.ActPos;
AxisOutput.Velocity:=Axis.NcToPlc.ActVelo;

END_FUNCTION_BLOCK

// ---- POUs/DrivingWheel2.TcPOU
FUNCTION_BLOCK DrivingWheel2
VAR_INPUT
	AxisInput:Command;//定义一个驱动轮PLC轴的输入结构体变量
END_VAR
VAR_OUTPUT
	AxisOutput:Status;//定义一个驱动轮PLC轴的输出结构体变量
END_VAR
VAR
	axis:axis_ref;		//定义一个轴
	power:mc_power;		//使能功能块
	moveAbsolute:mc_moveabsolute;//绝对运动功能块
	moveRelative:mc_moverelative;//相对运动功能块
	moveVelocity:mc_movevelocity;//匀速运动功能块
	reset:mc_reset;				//复位功能块
	halt:mc_halt;				//暂停功能块
	Home:mc_home;				//寻参功能块
	SetZero:mc_Setposition;		//强制设置位置功能块
	Dir: MC_Direction;			//匀速运动方向变量，1/3
	Signal:BOOL;				//寻参触发点
END_VAR

power(
	Axis:=axis, 
	Enable:=AxisInput.Enable, 
	Enable_Positive:=TRUE, 
	Enable_Negative:=TRUE, 
	Override:= , 
	BufferMode:= , 
	Options:= , 
	Status=>AxisOutput.Enable, 
	Busy=> , 
	Active=> , 
	Error=> , 
	ErrorID=> );
	
moveAbsolute(
	Axis:=axis, 
	Execute:=AxisInput.Move_Absolute, 
	Position:=AxisInput.Position, 
	Velocity:=AxisInput.Velocity, 
	Acceleration:= , 
	Deceleration:= , 
	Jerk:= , 
	BufferMode:= , 
	Options:= , 
	Done=> , 
	Busy=> , 
	Active=> , 
	CommandAborted=> , 
	Error=> , 
	ErrorID=> );

moveRelative(
	Axis:=axis, 
	Execute:=AxisInput.Move_Relative, 
	Distance:=AxisInput.Position, 
	Velocity:=AxisInput.Velocity, 
	Acceleration:= , 
	Deceleration:= , 
	Jerk:= , 
	BufferMode:= , 
	Options:= , 
	Done=> , 
	Busy=> , 
	Active=> , 
	CommandAborted=> , 
	Error=> , 
	ErrorID=> );

	IF(AxisInput.Velocity>=0)THEN
		Dir:=1;
	ELSIF(AxisInput.Velocity<0)THEN
		Dir:=3;
		AxisInput.Velocity:=-AxisInput.Velocity;
	END_IF
moveVelocity(
	Axis:= axis, 
	Execute:= AxisInput.Move_Velocity, 
	Velocity:= AxisInput.Velocity, 
	Acceleration:= , 
	Deceleration:= , 
	Jerk:= , 
	Direction:= Dir, 
	BufferMode:= , 
	Options:= , 
	InVelocity=> , 
	Busy=> , 
	Active=> , 
	CommandAborted=> , 
	Error=> , 
	ErrorID=> );
	
reset(
	Axis:= axis, 
	Execute:= AxisInput.Reset, 
	Done=> , 
	Busy=> , 
	Error=> , 
	ErrorID=> );
	
halt(
	Axis:= axis, 
	Execute:= AxisInput.Halt, 
	Deceleration:= , 
	Jerk:= , 
	BufferMode:= , 
	Options:= , 
	Done=> , 
	Busy=> , 
	Active=> , 
	CommandAborted=> , 
	Error=> , 
	ErrorID=> );
	IF(AxisInput.HomeSignal=524288)THEN
		Signal:=TRUE;
	ELSE 
		Signal:=FALSE;		
	END_IF	
Home(
	Axis:= axis, 
	Execute:= AxisInput.Home, 
	Position:= 0, 
	HomingMode:= , 
	BufferMode:= , 
	Options:= , 
	bCalibrationCam:= Signal, 
	Done=> , 
	Busy=> , 
	Active=> , 
	CommandAborted=> , 
	Error=> , 
	ErrorID=> );
	
SetZero(
	Axis:=axis , 
	Execute:=AxisInput.SetZero , 
	Position:= 0, 
	Mode:= , 
	Options:= , 
	Done=> , 
	Busy=> , 
	Error=> , 
	ErrorID=> );
AxisOutput.Position:=Axis.NcToPlc.ActPos;
AxisOutput.Velocity:=Axis.NcToPlc.ActVelo;

END_FUNCTION_BLOCK

// ---- POUs/DrivingWheel3.TcPOU
FUNCTION_BLOCK DrivingWheel3
VAR_INPUT
	AxisInput:Command;//定义一个驱动轮PLC轴的输入结构体变量
END_VAR
VAR_OUTPUT
	AxisOutput:Status;//定义一个驱动轮PLC轴的输出结构体变量
END_VAR
VAR
	axis:axis_ref;		//定义一个轴
	power:mc_power;		//使能功能块
	moveAbsolute:mc_moveabsolute;//绝对运动功能块
	moveRelative:mc_moverelative;//相对运动功能块
	moveVelocity:mc_movevelocity;//匀速运动功能块
	reset:mc_reset;				//复位功能块
	halt:mc_halt;				//暂停功能块
	Home:mc_home;				//寻参功能块
	SetZero:mc_Setposition;		//强制设置位置功能块
	Dir: MC_Direction;			//匀速运动方向变量，1/3
	Signal:BOOL;				//寻参触发点
END_VAR

power(
	Axis:=axis, 
	Enable:=AxisInput.Enable, 
	Enable_Positive:=TRUE, 
	Enable_Negative:=TRUE, 
	Override:= , 
	BufferMode:= , 
	Options:= , 
	Status=>AxisOutput.Enable, 
	Busy=> , 
	Active=> , 
	Error=> , 
	ErrorID=> );
	
moveAbsolute(
	Axis:=axis, 
	Execute:=AxisInput.Move_Absolute, 
	Position:=AxisInput.Position, 
	Velocity:=AxisInput.Velocity, 
	Acceleration:= , 
	Deceleration:= , 
	Jerk:= , 
	BufferMode:= , 
	Options:= , 
	Done=> , 
	Busy=> , 
	Active=> , 
	CommandAborted=> , 
	Error=> , 
	ErrorID=> );

moveRelative(
	Axis:=axis, 
	Execute:=AxisInput.Move_Relative, 
	Distance:=AxisInput.Position, 
	Velocity:=AxisInput.Velocity, 
	Acceleration:= , 
	Deceleration:= , 
	Jerk:= , 
	BufferMode:= , 
	Options:= , 
	Done=> , 
	Busy=> , 
	Active=> , 
	CommandAborted=> , 
	Error=> , 
	ErrorID=> );

	IF(AxisInput.Velocity>=0)THEN
		Dir:=1;
	ELSIF(AxisInput.Velocity<0)THEN
		Dir:=3;
		AxisInput.Velocity:=-AxisInput.Velocity;
	END_IF
moveVelocity(
	Axis:= axis, 
	Execute:= AxisInput.Move_Velocity, 
	Velocity:= AxisInput.Velocity, 
	Acceleration:= , 
	Deceleration:= , 
	Jerk:= , 
	Direction:= Dir, 
	BufferMode:= , 
	Options:= , 
	InVelocity=> , 
	Busy=> , 
	Active=> , 
	CommandAborted=> , 
	Error=> , 
	ErrorID=> );
	
reset(
	Axis:= axis, 
	Execute:= AxisInput.Reset, 
	Done=> , 
	Busy=> , 
	Error=> , 
	ErrorID=> );
	
halt(
	Axis:= axis, 
	Execute:= AxisInput.Halt, 
	Deceleration:= , 
	Jerk:= , 
	BufferMode:= , 
	Options:= , 
	Done=> , 
	Busy=> , 
	Active=> , 
	CommandAborted=> , 
	Error=> , 
	ErrorID=> );
	IF(AxisInput.HomeSignal=524288)THEN
		Signal:=TRUE;
	ELSE 
		Signal:=FALSE;		
	END_IF	
Home(
	Axis:= axis, 
	Execute:= AxisInput.Home, 
	Position:= 0, 
	HomingMode:= , 
	BufferMode:= , 
	Options:= , 
	bCalibrationCam:= Signal, 
	Done=> , 
	Busy=> , 
	Active=> , 
	CommandAborted=> , 
	Error=> , 
	ErrorID=> );
	
SetZero(
	Axis:=axis , 
	Execute:=AxisInput.SetZero , 
	Position:= 0, 
	Mode:= , 
	Options:= , 
	Done=> , 
	Busy=> , 
	Error=> , 
	ErrorID=> );
AxisOutput.Position:=Axis.NcToPlc.ActPos;
AxisOutput.Velocity:=Axis.NcToPlc.ActVelo;

END_FUNCTION_BLOCK

// ---- POUs/DrivingWheel4.TcPOU
FUNCTION_BLOCK DrivingWheel4
VAR_INPUT
	AxisInput:Command;//定义一个驱动轮PLC轴的输入结构体变量
END_VAR
VAR_OUTPUT
	AxisOutput:Status;//定义一个驱动轮PLC轴的输出结构体变量
END_VAR
VAR
	axis:axis_ref;		//定义一个轴
	power:mc_power;		//使能功能块
	moveAbsolute:mc_moveabsolute;//绝对运动功能块
	moveRelative:mc_moverelative;//相对运动功能块
	moveVelocity:mc_movevelocity;//匀速运动功能块
	reset:mc_reset;				//复位功能块
	halt:mc_halt;				//暂停功能块
	Home:mc_home;				//寻参功能块
	SetZero:mc_Setposition;		//强制设置位置功能块
	Dir: MC_Direction;			//匀速运动方向变量，1/3
	Signal:BOOL;				//寻参触发点
END_VAR

power(
	Axis:=axis, 
	Enable:=AxisInput.Enable, 
	Enable_Positive:=TRUE, 
	Enable_Negative:=TRUE, 
	Override:= , 
	BufferMode:= , 
	Options:= , 
	Status=>AxisOutput.Enable, 
	Busy=> , 
	Active=> , 
	Error=> , 
	ErrorID=> );
	
moveAbsolute(
	Axis:=axis, 
	Execute:=AxisInput.Move_Absolute, 
	Position:=AxisInput.Position, 
	Velocity:=AxisInput.Velocity, 
	Acceleration:= , 
	Deceleration:= , 
	Jerk:= , 
	BufferMode:= , 
	Options:= , 
	Done=> , 
	Busy=> , 
	Active=> , 
	CommandAborted=> , 
	Error=> , 
	ErrorID=> );

moveRelative(
	Axis:=axis, 
	Execute:=AxisInput.Move_Relative, 
	Distance:=AxisInput.Position, 
	Velocity:=AxisInput.Velocity, 
	Acceleration:= , 
	Deceleration:= , 
	Jerk:= , 
	BufferMode:= , 
	Options:= , 
	Done=> , 
	Busy=> , 
	Active=> , 
	CommandAborted=> , 
	Error=> , 
	ErrorID=> );

	IF(AxisInput.Velocity>=0)THEN
		Dir:=1;
	ELSIF(AxisInput.Velocity<0)THEN
		Dir:=3;
		AxisInput.Velocity:=-AxisInput.Velocity;
	END_IF
moveVelocity(
	Axis:= axis, 
	Execute:= AxisInput.Move_Velocity, 
	Velocity:= AxisInput.Velocity, 
	Acceleration:= , 
	Deceleration:= , 
	Jerk:= , 
	Direction:= Dir, 
	BufferMode:= , 
	Options:= , 
	InVelocity=> , 
	Busy=> , 
	Active=> , 
	CommandAborted=> , 
	Error=> , 
	ErrorID=> );
	
reset(
	Axis:= axis, 
	Execute:= AxisInput.Reset, 
	Done=> , 
	Busy=> , 
	Error=> , 
	ErrorID=> );
	
halt(
	Axis:= axis, 
	Execute:= AxisInput.Halt, 
	Deceleration:= , 
	Jerk:= , 
	BufferMode:= , 
	Options:= , 
	Done=> , 
	Busy=> , 
	Active=> , 
	CommandAborted=> , 
	Error=> , 
	ErrorID=> );
	IF(AxisInput.HomeSignal=524288)THEN
		Signal:=TRUE;
	ELSE 
		Signal:=FALSE;		
	END_IF	
Home(
	Axis:= axis, 
	Execute:= AxisInput.Home, 
	Position:= 0, 
	HomingMode:= , 
	BufferMode:= , 
	Options:= , 
	bCalibrationCam:= Signal, 
	Done=> , 
	Busy=> , 
	Active=> , 
	CommandAborted=> , 
	Error=> , 
	ErrorID=> );
	
SetZero(
	Axis:=axis , 
	Execute:=AxisInput.SetZero , 
	Position:= 0, 
	Mode:= , 
	Options:= , 
	Done=> , 
	Busy=> , 
	Error=> , 
	ErrorID=> );
AxisOutput.Position:=Axis.NcToPlc.ActPos;
AxisOutput.Velocity:=Axis.NcToPlc.ActVelo;

END_FUNCTION_BLOCK

// ---- POUs/SwingArm1.TcPOU
FUNCTION_BLOCK SwingArm1
VAR_INPUT
	AxisInput:Command;//定义一个驱动轮PLC轴的输入结构体变量
END_VAR
VAR_OUTPUT
	AxisOutput:Status;//定义一个驱动轮PLC轴的输出结构体变量
END_VAR
VAR
	axis:axis_ref;		//定义一个轴
	power:mc_power;		//使能功能块
	moveAbsolute:mc_moveabsolute;//绝对运动功能块
	moveRelative:mc_moverelative;//相对运动功能块
	moveVelocity:mc_movevelocity;//匀速运动功能块
	reset:mc_reset;				//复位功能块
	halt:mc_halt;				//暂停功能块
	Home:mc_home;				//寻参功能块
	SetZero:mc_Setposition;		//强制设置位置功能块
	Dir: MC_Direction;			//匀速运动方向变量，1/3
	Signal:BOOL;				//寻参触发点
END_VAR

power(
	Axis:=axis, 
	Enable:=AxisInput.Enable, 
	Enable_Positive:=TRUE, 
	Enable_Negative:=TRUE, 
	Override:= , 
	BufferMode:= , 
	Options:= , 
	Status=>AxisOutput.Enable, 
	Busy=> , 
	Active=> , 
	Error=> , 
	ErrorID=> );
	
moveAbsolute(
	Axis:=axis, 
	Execute:=AxisInput.Move_Absolute, 
	Position:=AxisInput.Position, 
	Velocity:=AxisInput.Velocity, 
	Acceleration:= , 
	Deceleration:= , 
	Jerk:= , 
	BufferMode:= , 
	Options:= , 
	Done=> , 
	Busy=> , 
	Active=> , 
	CommandAborted=> , 
	Error=> , 
	ErrorID=> );

moveRelative(
	Axis:=axis, 
	Execute:=AxisInput.Move_Relative, 
	Distance:=AxisInput.Position, 
	Velocity:=AxisInput.Velocity, 
	Acceleration:= , 
	Deceleration:= , 
	Jerk:= , 
	BufferMode:= , 
	Options:= , 
	Done=> , 
	Busy=> , 
	Active=> , 
	CommandAborted=> , 
	Error=> , 
	ErrorID=> );

	IF(AxisInput.Velocity>=0)THEN
		Dir:=1;
	ELSIF(AxisInput.Velocity<0)THEN
		Dir:=3;
		AxisInput.Velocity:=-AxisInput.Velocity;
	END_IF
moveVelocity(
	Axis:= axis, 
	Execute:= AxisInput.Move_Velocity, 
	Velocity:= AxisInput.Velocity, 
	Acceleration:= , 
	Deceleration:= , 
	Jerk:= , 
	Direction:= Dir, 
	BufferMode:= , 
	Options:= , 
	InVelocity=> , 
	Busy=> , 
	Active=> , 
	CommandAborted=> , 
	Error=> , 
	ErrorID=> );
	
reset(
	Axis:= axis, 
	Execute:= AxisInput.Reset, 
	Done=> , 
	Busy=> , 
	Error=> , 
	ErrorID=> );
	
halt(
	Axis:= axis, 
	Execute:= AxisInput.Halt, 
	Deceleration:= , 
	Jerk:= , 
	BufferMode:= , 
	Options:= , 
	Done=> , 
	Busy=> , 
	Active=> , 
	CommandAborted=> , 
	Error=> , 
	ErrorID=> );
	IF(AxisInput.HomeSignal=524288)THEN
		Signal:=TRUE;
	ELSE 
		Signal:=FALSE;		
	END_IF	
Home(
	Axis:= axis, 
	Execute:= AxisInput.Home, 
	Position:= 0, 
	HomingMode:= , 
	BufferMode:= , 
	Options:= , 
	bCalibrationCam:= Signal, 
	Done=> , 
	Busy=> , 
	Active=> , 
	CommandAborted=> , 
	Error=> , 
	ErrorID=> );
	
SetZero(
	Axis:=axis , 
	Execute:=AxisInput.SetZero , 
	Position:= 0, 
	Mode:= , 
	Options:= , 
	Done=> , 
	Busy=> , 
	Error=> , 
	ErrorID=> );
AxisOutput.Position:=Axis.NcToPlc.ActPos-90;
AxisOutput.Velocity:=Axis.NcToPlc.ActVelo;

END_FUNCTION_BLOCK

// ---- POUs/SwingArm2.TcPOU
FUNCTION_BLOCK SwingArm2
VAR_INPUT
	AxisInput:Command;//定义一个驱动轮PLC轴的输入结构体变量
END_VAR
VAR_OUTPUT
	AxisOutput:Status;//定义一个驱动轮PLC轴的输出结构体变量
END_VAR
VAR
	axis:axis_ref;		//定义一个轴
	power:mc_power;		//使能功能块
	moveAbsolute:mc_moveabsolute;//绝对运动功能块
	moveRelative:mc_moverelative;//相对运动功能块
	moveVelocity:mc_movevelocity;//匀速运动功能块
	reset:mc_reset;				//复位功能块
	halt:mc_halt;				//暂停功能块
	Home:mc_home;				//寻参功能块
	SetZero:mc_Setposition;		//强制设置位置功能块
	Dir: MC_Direction;			//匀速运动方向变量，1/3
	Signal:BOOL;				//寻参触发点
END_VAR

power(
	Axis:=axis, 
	Enable:=AxisInput.Enable, 
	Enable_Positive:=TRUE, 
	Enable_Negative:=TRUE, 
	Override:= , 
	BufferMode:= , 
	Options:= , 
	Status=>AxisOutput.Enable, 
	Busy=> , 
	Active=> , 
	Error=> , 
	ErrorID=> );
	
moveAbsolute(
	Axis:=axis, 
	Execute:=AxisInput.Move_Absolute, 
	Position:=AxisInput.Position, 
	Velocity:=AxisInput.Velocity, 
	Acceleration:= , 
	Deceleration:= , 
	Jerk:= , 
	BufferMode:= , 
	Options:= , 
	Done=> , 
	Busy=> , 
	Active=> , 
	CommandAborted=> , 
	Error=> , 
	ErrorID=> );

moveRelative(
	Axis:=axis, 
	Execute:=AxisInput.Move_Relative, 
	Distance:=AxisInput.Position, 
	Velocity:=AxisInput.Velocity, 
	Acceleration:= , 
	Deceleration:= , 
	Jerk:= , 
	BufferMode:= , 
	Options:= , 
	Done=> , 
	Busy=> , 
	Active=> , 
	CommandAborted=> , 
	Error=> , 
	ErrorID=> );

	IF(AxisInput.Velocity>=0)THEN
		Dir:=1;
	ELSIF(AxisInput.Velocity<0)THEN
		Dir:=3;
		AxisInput.Velocity:=-AxisInput.Velocity;
	END_IF
moveVelocity(
	Axis:= axis, 
	Execute:= AxisInput.Move_Velocity, 
	Velocity:= AxisInput.Velocity, 
	Acceleration:= , 
	Deceleration:= , 
	Jerk:= , 
	Direction:= Dir, 
	BufferMode:= , 
	Options:= , 
	InVelocity=> , 
	Busy=> , 
	Active=> , 
	CommandAborted=> , 
	Error=> , 
	ErrorID=> );
	
reset(
	Axis:= axis, 
	Execute:= AxisInput.Reset, 
	Done=> , 
	Busy=> , 
	Error=> , 
	ErrorID=> );
	
halt(
	Axis:= axis, 
	Execute:= AxisInput.Halt, 
	Deceleration:= , 
	Jerk:= , 
	BufferMode:= , 
	Options:= , 
	Done=> , 
	Busy=> , 
	Active=> , 
	CommandAborted=> , 
	Error=> , 
	ErrorID=> );
	IF(AxisInput.HomeSignal=524288)THEN
		Signal:=TRUE;
	ELSE 
		Signal:=FALSE;		
	END_IF	
Home(
	Axis:= axis, 
	Execute:= AxisInput.Home, 
	Position:= 0, 
	HomingMode:= , 
	BufferMode:= , 
	Options:= , 
	bCalibrationCam:= Signal, 
	Done=> , 
	Busy=> , 
	Active=> , 
	CommandAborted=> , 
	Error=> , 
	ErrorID=> );
	
SetZero(
	Axis:=axis , 
	Execute:=AxisInput.SetZero , 
	Position:= 0, 
	Mode:= , 
	Options:= , 
	Done=> , 
	Busy=> , 
	Error=> , 
	ErrorID=> );
AxisOutput.Position:=Axis.NcToPlc.ActPos-90;
AxisOutput.Velocity:=Axis.NcToPlc.ActVelo;

END_FUNCTION_BLOCK

// ---- POUs/SwingArm3.TcPOU
FUNCTION_BLOCK SwingArm3
VAR_INPUT
	AxisInput:Command;//定义一个驱动轮PLC轴的输入结构体变量
END_VAR
VAR_OUTPUT
	AxisOutput:Status;//定义一个驱动轮PLC轴的输出结构体变量
END_VAR
VAR
	axis:axis_ref;		//定义一个轴
	power:mc_power;		//使能功能块
	moveAbsolute:mc_moveabsolute;//绝对运动功能块
	moveRelative:mc_moverelative;//相对运动功能块
	moveVelocity:mc_movevelocity;//匀速运动功能块
	reset:mc_reset;				//复位功能块
	halt:mc_halt;				//暂停功能块
	Home:mc_home;				//寻参功能块
	SetZero:mc_Setposition;		//强制设置位置功能块
	Dir: MC_Direction;			//匀速运动方向变量，1/3
	Signal:BOOL;				//寻参触发点
END_VAR

power(
	Axis:=axis, 
	Enable:=AxisInput.Enable, 
	Enable_Positive:=TRUE, 
	Enable_Negative:=TRUE, 
	Override:= , 
	BufferMode:= , 
	Options:= , 
	Status=>AxisOutput.Enable, 
	Busy=> , 
	Active=> , 
	Error=> , 
	ErrorID=> );
	
moveAbsolute(
	Axis:=axis, 
	Execute:=AxisInput.Move_Absolute, 
	Position:=AxisInput.Position, 
	Velocity:=AxisInput.Velocity, 
	Acceleration:= , 
	Deceleration:= , 
	Jerk:= , 
	BufferMode:= , 
	Options:= , 
	Done=> , 
	Busy=> , 
	Active=> , 
	CommandAborted=> , 
	Error=> , 
	ErrorID=> );

moveRelative(
	Axis:=axis, 
	Execute:=AxisInput.Move_Relative, 
	Distance:=AxisInput.Position, 
	Velocity:=AxisInput.Velocity, 
	Acceleration:= , 
	Deceleration:= , 
	Jerk:= , 
	BufferMode:= , 
	Options:= , 
	Done=> , 
	Busy=> , 
	Active=> , 
	CommandAborted=> , 
	Error=> , 
	ErrorID=> );

	IF(AxisInput.Velocity>=0)THEN
		Dir:=1;
	ELSIF(AxisInput.Velocity<0)THEN
		Dir:=3;
		AxisInput.Velocity:=-AxisInput.Velocity;
	END_IF
moveVelocity(
	Axis:= axis, 
	Execute:= AxisInput.Move_Velocity, 
	Velocity:= AxisInput.Velocity, 
	Acceleration:= , 
	Deceleration:= , 
	Jerk:= , 
	Direction:= Dir, 
	BufferMode:= , 
	Options:= , 
	InVelocity=> , 
	Busy=> , 
	Active=> , 
	CommandAborted=> , 
	Error=> , 
	ErrorID=> );
	
reset(
	Axis:= axis, 
	Execute:= AxisInput.Reset, 
	Done=> , 
	Busy=> , 
	Error=> , 
	ErrorID=> );
	
halt(
	Axis:= axis, 
	Execute:= AxisInput.Halt, 
	Deceleration:= , 
	Jerk:= , 
	BufferMode:= , 
	Options:= , 
	Done=> , 
	Busy=> , 
	Active=> , 
	CommandAborted=> , 
	Error=> , 
	ErrorID=> );
	IF(AxisInput.HomeSignal=524288)THEN
		Signal:=TRUE;
	ELSE 
		Signal:=FALSE;		
	END_IF	
Home(
	Axis:= axis, 
	Execute:= AxisInput.Home, 
	Position:= 0, 
	HomingMode:= , 
	BufferMode:= , 
	Options:= , 
	bCalibrationCam:= Signal, 
	Done=> , 
	Busy=> , 
	Active=> , 
	CommandAborted=> , 
	Error=> , 
	ErrorID=> );
	
SetZero(
	Axis:=axis , 
	Execute:=AxisInput.SetZero , 
	Position:= 0, 
	Mode:= , 
	Options:= , 
	Done=> , 
	Busy=> , 
	Error=> , 
	ErrorID=> );
AxisOutput.Position:=Axis.NcToPlc.ActPos-90;
AxisOutput.Velocity:=Axis.NcToPlc.ActVelo;

END_FUNCTION_BLOCK

// ---- POUs/SwingArm4.TcPOU
FUNCTION_BLOCK SwingArm4
VAR_INPUT
	AxisInput:Command;//定义一个驱动轮PLC轴的输入结构体变量
END_VAR
VAR_OUTPUT
	AxisOutput:Status;//定义一个驱动轮PLC轴的输出结构体变量
END_VAR
VAR
	axis:axis_ref;		//定义一个轴
	power:mc_power;		//使能功能块
	moveAbsolute:mc_moveabsolute;//绝对运动功能块
	moveRelative:mc_moverelative;//相对运动功能块
	moveVelocity:mc_movevelocity;//匀速运动功能块
	reset:mc_reset;				//复位功能块
	halt:mc_halt;				//暂停功能块
	Home:mc_home;				//寻参功能块
	SetZero:mc_Setposition;		//强制设置位置功能块
	Dir: MC_Direction;			//匀速运动方向变量，1/3
	Signal:BOOL;				//寻参触发点
END_VAR

power(
	Axis:=axis, 
	Enable:=AxisInput.Enable, 
	Enable_Positive:=TRUE, 
	Enable_Negative:=TRUE, 
	Override:= , 
	BufferMode:= , 
	Options:= , 
	Status=>AxisOutput.Enable, 
	Busy=> , 
	Active=> , 
	Error=> , 
	ErrorID=> );
	
moveAbsolute(
	Axis:=axis, 
	Execute:=AxisInput.Move_Absolute, 
	Position:=AxisInput.Position, 
	Velocity:=AxisInput.Velocity, 
	Acceleration:= , 
	Deceleration:= , 
	Jerk:= , 
	BufferMode:= , 
	Options:= , 
	Done=> , 
	Busy=> , 
	Active=> , 
	CommandAborted=> , 
	Error=> , 
	ErrorID=> );

moveRelative(
	Axis:=axis, 
	Execute:=AxisInput.Move_Relative, 
	Distance:=AxisInput.Position, 
	Velocity:=AxisInput.Velocity, 
	Acceleration:= , 
	Deceleration:= , 
	Jerk:= , 
	BufferMode:= , 
	Options:= , 
	Done=> , 
	Busy=> , 
	Active=> , 
	CommandAborted=> , 
	Error=> , 
	ErrorID=> );

	IF(AxisInput.Velocity>=0)THEN
		Dir:=1;
	ELSIF(AxisInput.Velocity<0)THEN
		Dir:=3;
		AxisInput.Velocity:=-AxisInput.Velocity;
	END_IF
moveVelocity(
	Axis:= axis, 
	Execute:= AxisInput.Move_Velocity, 
	Velocity:= AxisInput.Velocity, 
	Acceleration:= , 
	Deceleration:= , 
	Jerk:= , 
	Direction:= Dir, 
	BufferMode:= , 
	Options:= , 
	InVelocity=> , 
	Busy=> , 
	Active=> , 
	CommandAborted=> , 
	Error=> , 
	ErrorID=> );
	
reset(
	Axis:= axis, 
	Execute:= AxisInput.Reset, 
	Done=> , 
	Busy=> , 
	Error=> , 
	ErrorID=> );
	
halt(
	Axis:= axis, 
	Execute:= AxisInput.Halt, 
	Deceleration:= , 
	Jerk:= , 
	BufferMode:= , 
	Options:= , 
	Done=> , 
	Busy=> , 
	Active=> , 
	CommandAborted=> , 
	Error=> , 
	ErrorID=> );
	IF(AxisInput.HomeSignal=524288)THEN
		Signal:=TRUE;
	ELSE 
		Signal:=FALSE;		
	END_IF	
Home(
	Axis:= axis, 
	Execute:= AxisInput.Home, 
	Position:= 0, 
	HomingMode:= , 
	BufferMode:= , 
	Options:= , 
	bCalibrationCam:= Signal, 
	Done=> , 
	Busy=> , 
	Active=> , 
	CommandAborted=> , 
	Error=> , 
	ErrorID=> );
	
SetZero(
	Axis:=axis , 
	Execute:=AxisInput.SetZero , 
	Position:= 0, 
	Mode:= , 
	Options:= , 
	Done=> , 
	Busy=> , 
	Error=> , 
	ErrorID=> );
AxisOutput.Position:=Axis.NcToPlc.ActPos-90;
AxisOutput.Velocity:=Axis.NcToPlc.ActVelo;

END_FUNCTION_BLOCK

// ---- POUs/Waist.TcPOU
FUNCTION_BLOCK Waist
VAR_INPUT
	AxisInput:Command;//定义一个驱动轮PLC轴的输入结构体变量
END_VAR
VAR_OUTPUT
	AxisOutput:Status;//定义一个驱动轮PLC轴的输出结构体变量
END_VAR
VAR
	axis:axis_ref;		//定义一个轴
	power:mc_power;		//使能功能块
	moveAbsolute:mc_moveabsolute;//绝对运动功能块
	moveRelative:mc_moverelative;//相对运动功能块
	moveVelocity:mc_movevelocity;//匀速运动功能块
	reset:mc_reset;				//复位功能块
	halt:mc_halt;				//暂停功能块
	Home:mc_home;				//寻参功能块
	SetZero:mc_Setposition;		//强制设置位置功能块
	Dir: MC_Direction;			//匀速运动方向变量，1/3
	Signal:BOOL;				//寻参触发点
END_VAR

power(
	Axis:=axis, 
	Enable:=AxisInput.Enable, 
	Enable_Positive:=TRUE, 
	Enable_Negative:=TRUE, 
	Override:= , 
	BufferMode:= , 
	Options:= , 
	Status=>AxisOutput.Enable, 
	Busy=> , 
	Active=> , 
	Error=> , 
	ErrorID=> );
	
moveAbsolute(
	Axis:=axis, 
	Execute:=AxisInput.Move_Absolute, 
	Position:=AxisInput.Position, 
	Velocity:=AxisInput.Velocity, 
	Acceleration:= , 
	Deceleration:= , 
	Jerk:= , 
	BufferMode:= , 
	Options:= , 
	Done=> , 
	Busy=> , 
	Active=> , 
	CommandAborted=> , 
	Error=> , 
	ErrorID=> );

moveRelative(
	Axis:=axis, 
	Execute:=AxisInput.Move_Relative, 
	Distance:=AxisInput.Position, 
	Velocity:=AxisInput.Velocity, 
	Acceleration:= , 
	Deceleration:= , 
	Jerk:= , 
	BufferMode:= , 
	Options:= , 
	Done=> , 
	Busy=> , 
	Active=> , 
	CommandAborted=> , 
	Error=> , 
	ErrorID=> );

	IF(AxisInput.Velocity>=0)THEN
		Dir:=1;
	ELSIF(AxisInput.Velocity<0)THEN
		Dir:=3;
		AxisInput.Velocity:=-AxisInput.Velocity;
	END_IF
moveVelocity(
	Axis:= axis, 
	Execute:= AxisInput.Move_Velocity, 
	Velocity:= AxisInput.Velocity, 
	Acceleration:= , 
	Deceleration:= , 
	Jerk:= , 
	Direction:= Dir, 
	BufferMode:= , 
	Options:= , 
	InVelocity=> , 
	Busy=> , 
	Active=> , 
	CommandAborted=> , 
	Error=> , 
	ErrorID=> );
	
reset(
	Axis:= axis, 
	Execute:= AxisInput.Reset, 
	Done=> , 
	Busy=> , 
	Error=> , 
	ErrorID=> );
	
halt(
	Axis:= axis, 
	Execute:= AxisInput.Halt, 
	Deceleration:= , 
	Jerk:= , 
	BufferMode:= , 
	Options:= , 
	Done=> , 
	Busy=> , 
	Active=> , 
	CommandAborted=> , 
	Error=> , 
	ErrorID=> );
	IF(AxisInput.HomeSignal=524288)THEN
		Signal:=TRUE;
	ELSE 
		Signal:=FALSE;		
	END_IF	
Home(
	Axis:= axis, 
	Execute:= AxisInput.Home, 
	Position:= 0, 
	HomingMode:= , 
	BufferMode:= , 
	Options:= , 
	bCalibrationCam:= Signal, 
	Done=> , 
	Busy=> , 
	Active=> , 
	CommandAborted=> , 
	Error=> , 
	ErrorID=> );
	
SetZero(
	Axis:=axis , 
	Execute:=AxisInput.SetZero , 
	Position:= 0, 
	Mode:= , 
	Options:= , 
	Done=> , 
	Busy=> , 
	Error=> , 
	ErrorID=> );
AxisOutput.Position:=Axis.NcToPlc.ActPos;
AxisOutput.Velocity:=Axis.NcToPlc.ActVelo;

END_FUNCTION_BLOCK

// ---- POUs/BigArm.TcPOU
FUNCTION_BLOCK BigArm
VAR_INPUT
	AxisInput:Command;//定义一个驱动轮PLC轴的输入结构体变量
END_VAR
VAR_OUTPUT
	AxisOutput:Status;//定义一个驱动轮PLC轴的输出结构体变量
END_VAR
VAR
	axis:axis_ref;		//定义一个轴
	power:mc_power;		//使能功能块
	moveAbsolute:mc_moveabsolute;//绝对运动功能块
	moveRelative:mc_moverelative;//相对运动功能块
	moveVelocity:mc_movevelocity;//匀速运动功能块
	reset:mc_reset;				//复位功能块
	halt:mc_halt;				//暂停功能块
	Home:mc_home;				//寻参功能块
	SetZero:mc_Setposition;		//强制设置位置功能块
	Dir: MC_Direction;			//匀速运动方向变量，1/3
	Signal:BOOL;				//寻参触发点
	temp:LREAL;
	flag: INT:=0;
	start_flag: BOOL:=TRUE;
	start_position: LREAL;
	moveRelative_do: BOOL;
	temp_position: LREAL;
	temp_velocity: LREAL;
	coefficient:INT:=1;
END_VAR

IF Axis.NcToPlc.ActPos-74.9>180 THEN
	temp:=360;
ELSIF Axis.NcToPlc.ActPos-74.9<-180	THEN
	temp:=-360;
ELSE
	temp:=0;		
END_IF
AxisOutput.Position:=Axis.NcToPlc.ActPos-74.9-temp;
IF start_flag THEN
	start_position:=AxisOutput.Position;
	start_flag:=FALSE;
END_IF
IF AxisOutput.Enable=FALSE THEN
	start_flag:=TRUE;
END_IF
IF start_position-1>0 THEN 
	coefficient:=-1;
ELSE 
	coefficient:=1;
END_IF
GVL.bigarm_position:=start_position;
AxisOutput.Velocity:=Axis.NcToPlc.ActVelo;
power(
	Axis:=axis, 
	Enable:=AxisInput.Enable, 
	Enable_Positive:=TRUE, 
	Enable_Negative:=TRUE, 
	Override:= , 
	BufferMode:= , 
	Options:= ,                   
	Status=>AxisOutput.Enable, 
	Busy=> , 
	Active=> , 
	Error=> , 
	ErrorID=> );
	
IF 	AxisOutput.Enable AND flag=0 THEN
	moveRelative_do:=TRUE;
	temp_position:=0.3*coefficient;
	temp_velocity:=1;
	flag:=1;
END_IF
IF flag=1 AND (AxisOutput.Position-start_position)*coefficient>0.2 THEN
	moveRelative_do:=AxisInput.Move_Relative;
	temp_position:=AxisInput.Position;
	temp_velocity:=AxisInput.Velocity;
	flag:=2;
END_IF
IF AxisOutput.Enable=FALSE AND flag=2 THEN
	flag:=0;
END_IF	
moveAbsolute(
	Axis:=axis, 
	Execute:=AxisInput.Move_Absolute, 
	Position:=AxisInput.Position+74.9+temp, 
	Velocity:=AxisInput.Velocity, 
	Acceleration:= , 
	Deceleration:= , 
	Jerk:= , 
	BufferMode:= , 
	Options:= , 
	Done=> , 
	Busy=> , 
	Active=> , 
	CommandAborted=> , 
	Error=> , 
	ErrorID=> );
moveRelative(
	Axis:=axis, 
	Execute:=moveRelative_do, 
	Distance:=temp_position, 
	Velocity:=temp_velocity, 
	Acceleration:= , 
	Deceleration:= , 
	Jerk:= , 
	BufferMode:= , 
	Options:= , 
	Done=> , 
	Busy=> , 
	Active=> , 
	CommandAborted=> , 
	Error=> , 
	ErrorID=> );

	IF(AxisInput.Velocity>=0)THEN
		Dir:=1;
	ELSIF(AxisInput.Velocity<0)THEN
		Dir:=3;
		AxisInput.Velocity:=-AxisInput.Velocity;
	END_IF
moveVelocity(
	Axis:= axis, 
	Execute:= AxisInput.Move_Velocity, 
	Velocity:= AxisInput.Velocity, 
	Acceleration:= , 
	Deceleration:= , 
	Jerk:= , 
	Direction:= Dir, 
	BufferMode:= , 
	Options:= , 
	InVelocity=> , 
	Busy=> , 
	Active=> , 
	CommandAborted=> , 
	Error=> , 
	ErrorID=> );
	
reset(
	Axis:= axis, 
	Execute:= AxisInput.Reset, 
	Done=> , 
	Busy=> , 
	Error=> , 
	ErrorID=> );
	
halt(
	Axis:= axis, 
	Execute:= AxisInput.Halt, 
	Deceleration:= , 
	Jerk:= , 
	BufferMode:= , 
	Options:= , 
	Done=> , 
	Busy=> , 
	Active=> , 
	CommandAborted=> , 
	Error=> , 
	ErrorID=> );
	IF(AxisInput.HomeSignal=524288)THEN
		Signal:=TRUE;
	ELSE 
		Signal:=FALSE;		
	END_IF	
Home(
	Axis:= axis, 
	Execute:= AxisInput.Home, 
	Position:= 0, 
	HomingMode:= , 
	BufferMode:= , 
	Options:= , 
	bCalibrationCam:= Signal, 
	Done=> , 
	Busy=> , 
	Active=> , 
	CommandAborted=> , 
	Error=> , 
	ErrorID=> );
	
SetZero(
	Axis:=axis , 
	Execute:=AxisInput.SetZero , 
	Position:= 0, 
	Mode:= , 
	Options:= , 
	Done=> , 
	Busy=> , 
	Error=> , 
	ErrorID=> );

END_FUNCTION_BLOCK

// ---- POUs/Flex.TcPOU
FUNCTION_BLOCK Flex
VAR_INPUT
	AxisInput:Command;//定义一个驱动轮PLC轴的输入结构体变量
END_VAR
VAR_OUTPUT
	AxisOutput:Status;//定义一个驱动轮PLC轴的输出结构体变量
END_VAR
VAR
	axis:axis_ref;		//定义一个轴
	power:mc_power;		//使能功能块
	moveAbsolute:mc_moveabsolute;//绝对运动功能块
	moveRelative:mc_moverelative;//相对运动功能块
	moveVelocity:mc_movevelocity;//匀速运动功能块
	reset:mc_reset;				//复位功能块
	halt:mc_halt;				//暂停功能块
	Home:mc_home;				//寻参功能块
	SetZero:mc_Setposition;		//强制设置位置功能块
	Dir: MC_Direction;			//匀速运动方向变量，1/3
	Signal:BOOL;				//寻参触发点
END_VAR

power(
	Axis:=axis, 
	Enable:=AxisInput.Enable, 
	Enable_Positive:=TRUE, 
	Enable_Negative:=TRUE, 
	Override:= , 
	BufferMode:= , 
	Options:= , 
	Status=>AxisOutput.Enable, 
	Busy=> , 
	Active=> , 
	Error=> , 
	ErrorID=> );
	
moveAbsolute(
	Axis:=axis, 
	Execute:=AxisInput.Move_Absolute, 
	Position:=AxisInput.Position, 
	Velocity:=AxisInput.Velocity, 
	Acceleration:= , 
	Deceleration:= , 
	Jerk:= , 
	BufferMode:= , 
	Options:= , 
	Done=> , 
	Busy=> , 
	Active=> , 
	CommandAborted=> , 
	Error=> , 
	ErrorID=> );

moveRelative(
	Axis:=axis, 
	Execute:=AxisInput.Move_Relative, 
	Distance:=AxisInput.Position, 
	Velocity:=AxisInput.Velocity, 
	Acceleration:= , 
	Deceleration:= , 
	Jerk:= , 
	BufferMode:= , 
	Options:= , 
	Done=> , 
	Busy=> , 
	Active=> , 
	CommandAborted=> , 
	Error=> , 
	ErrorID=> );

	IF(AxisInput.Velocity>=0)THEN
		Dir:=1;
	ELSIF(AxisInput.Velocity<0)THEN
		Dir:=3;
		AxisInput.Velocity:=-AxisInput.Velocity;
	END_IF
moveVelocity(
	Axis:= axis, 
	Execute:= AxisInput.Move_Velocity, 
	Velocity:= AxisInput.Velocity, 
	Acceleration:= , 
	Deceleration:= , 
	Jerk:= , 
	Direction:= Dir, 
	BufferMode:= , 
	Options:= , 
	InVelocity=> , 
	Busy=> , 
	Active=> , 
	CommandAborted=> , 
	Error=> , 
	ErrorID=> );
	
reset(
	Axis:= axis, 
	Execute:= AxisInput.Reset, 
	Done=> , 
	Busy=> , 
	Error=> , 
	ErrorID=> );
	
halt(
	Axis:= axis, 
	Execute:= AxisInput.Halt, 
	Deceleration:= , 
	Jerk:= , 
	BufferMode:= , 
	Options:= , 
	Done=> , 
	Busy=> , 
	Active=> , 
	CommandAborted=> , 
	Error=> , 
	ErrorID=> );
	IF(AxisInput.HomeSignal=524288)THEN
		Signal:=TRUE;
	ELSE 
		Signal:=FALSE;		
	END_IF	
Home(
	Axis:= axis, 
	Execute:= AxisInput.Home, 
	Position:= 0, 
	HomingMode:= , 
	BufferMode:= , 
	Options:= , 
	bCalibrationCam:= Signal, 
	Done=> , 
	Busy=> , 
	Active=> , 
	CommandAborted=> , 
	Error=> , 
	ErrorID=> );
	
SetZero(
	Axis:=axis , 
	Execute:=AxisInput.SetZero , 
	Position:= 0, 
	Mode:= , 
	Options:= , 
	Done=> , 
	Busy=> , 
	Error=> , 
	ErrorID=> );
AxisOutput.Position:=Axis.NcToPlc.ActPos;
AxisOutput.Velocity:=Axis.NcToPlc.ActVelo;

END_FUNCTION_BLOCK

// ---- POUs/MiddleArm.TcPOU
FUNCTION_BLOCK MiddleArm
VAR_INPUT
	AxisInput:Command;//定义一个驱动轮PLC轴的输入结构体变量
END_VAR
VAR_OUTPUT
	AxisOutput:Status;//定义一个驱动轮PLC轴的输出结构体变量
END_VAR
VAR
	axis:axis_ref;		//定义一个轴
	power:mc_power;		//使能功能块
	moveAbsolute:mc_moveabsolute;//绝对运动功能块
	moveRelative:mc_moverelative;//相对运动功能块
	moveVelocity:mc_movevelocity;//匀速运动功能块
	reset:mc_reset;				//复位功能块
	halt:mc_halt;				//暂停功能块
	Home:mc_home;				//寻参功能块
	SetZero:mc_Setposition;		//强制设置位置功能块
	Dir: MC_Direction;			//匀速运动方向变量，1/3
	Signal:BOOL;				//寻参触发点
	Halt_do: BOOL;
	mode: MC_HomingMode;
	temp:LREAL;
	flag: INT:=0;
	moveRelative_do: BOOL;
	temp_position: LREAL;
	temp_velocity: LREAL;
	start_position:LREAL;
	start_flag:BOOL:=TRUE;
	coefficient:INT:=1;
END_VAR

IF Axis.NcToPlc.ActPos-16.3>180 THEN
	temp:=360;
ELSIF Axis.NcToPlc.ActPos-16.3<-180	THEN
	temp:=-360;
ELSE
	temp:=0;		
END_IF
AxisOutput.Position:=Axis.NcToPlc.ActPos-16.3-temp;
IF start_flag THEN
	start_position:=AxisOutput.Position;
	start_flag:=FALSE;
END_IF
IF AxisOutput.Enable=FALSE THEN
	start_flag:=TRUE;
END_IF
GVL.middlearm_position:=start_position;
GVL.middlearm_position:=GVL.bigarm_position+GVL.middlearm_position;
IF GVL.middlearm_position-1>0 THEN 
	coefficient:=-1;
ELSE 
	coefficient:=1;
END_IF
AxisOutput.Velocity:=Axis.NcToPlc.ActVelo;
power(
	Axis:=axis, 
	Enable:=AxisInput.Enable, 
	Enable_Positive:=TRUE, 
	Enable_Negative:=TRUE, 
	Override:= , 
	BufferMode:= , 
	Options:= , 
	Status=>AxisOutput.Enable, 
	Busy=> , 
	Active=> , 
	Error=> , 
	ErrorID=> );
IF 	AxisOutput.Enable AND flag=0 THEN
	moveRelative_do:=TRUE;
	temp_position:=0.3*coefficient;
	temp_velocity:=1;
	flag:=1;
END_IF
IF flag=1 AND (AxisOutput.Position-start_position)*coefficient>0.2 THEN
	moveRelative_do:=AxisInput.Move_Relative;
	temp_position:=AxisInput.Position;
	temp_velocity:=AxisInput.Velocity;
	flag:=2;
END_IF
IF AxisOutput.Enable=FALSE AND flag=2 THEN
	flag:=0;
END_IF	
moveAbsolute(
	Axis:=axis, 
	Execute:=AxisInput.Move_Absolute, 
	Position:=AxisInput.Position+16.3+temp, 
	Velocity:=AxisInput.Velocity, 
	Acceleration:= , 
	Deceleration:= , 
	Jerk:= , 
	BufferMode:= , 
	Options:= , 
	Done=> , 
	Busy=> , 
	Active=> , 
	CommandAborted=> , 
	Error=> , 
	ErrorID=> );

moveRelative(
	Axis:=axis, 
	Execute:=moveRelative_do, 
	Distance:=temp_position, 
	Velocity:=temp_velocity, 
	Acceleration:= , 
	Deceleration:= , 
	Jerk:= , 
	BufferMode:= , 
	Options:= , 
	Done=> , 
	Busy=> , 
	Active=> , 
	CommandAborted=> , 
	Error=> , 
	ErrorID=> );

	IF(AxisInput.Velocity>=0)THEN
		Dir:=1;
	ELSIF(AxisInput.Velocity<0)THEN
		Dir:=3;
		AxisInput.Velocity:=-AxisInput.Velocity;
	END_IF
moveVelocity(
	Axis:= axis, 
	Execute:= AxisInput.Move_Velocity, 
	Velocity:= AxisInput.Velocity, 
	Acceleration:= , 
	Deceleration:= , 
	Jerk:= , 
	Direction:= Dir, 
	BufferMode:= , 
	Options:= , 
	InVelocity=> , 
	Busy=> , 
	Active=> , 
	CommandAborted=> , 
	Error=> , 
	ErrorID=> );
	
reset(
	Axis:= axis, 
	Execute:= AxisInput.Reset, 
	Done=> , 
	Busy=> , 
	Error=> , 
	ErrorID=> );
halt(
	Axis:= axis, 
	Execute:=AxisInput.Halt, 
	Deceleration:= , 
	Jerk:= , 
	BufferMode:= , 
	Options:= , 
	Done=> , 
	Busy=> , 
	Active=> , 
	CommandAborted=> , 
	Error=> , 
	ErrorID=> );
	IF(AxisInput.HomeSignal=524296)THEN
		Signal:=TRUE;
	ELSE 
		Signal:=FALSE;		
	END_IF	
Home(
	Axis:= axis, 
	Execute:= AxisInput.Home, 
	Position:= 0, 
	HomingMode:= , 
	BufferMode:= , 
	Options:= , 
	bCalibrationCam:= Signal, 
	Done=> , 
	Busy=> , 
	Active=> , 
	CommandAborted=> , 
	Error=> , 
	ErrorID=> );
	
SetZero(
	Axis:=axis , 
	Execute:=AxisInput.SetZero , 
	Position:= 0, 
	Mode:= , 
	Options:= , 
	Done=> , 
	Busy=> , 
	Error=> , 
	ErrorID=> );

END_FUNCTION_BLOCK

// ---- POUs/SmallArm.TcPOU
FUNCTION_BLOCK SmallArm
VAR_INPUT
	AxisInput:Command;//定义一个驱动轮PLC轴的输入结构体变量
END_VAR
VAR_OUTPUT
	AxisOutput:Status;//定义一个驱动轮PLC轴的输出结构体变量
END_VAR
VAR
	axis:axis_ref;		//定义一个轴
	power:mc_power;		//使能功能块
	moveAbsolute:mc_moveabsolute;//绝对运动功能块
	moveRelative:mc_moverelative;//相对运动功能块
	moveVelocity:mc_movevelocity;//匀速运动功能块
	reset:mc_reset;				//复位功能块
	halt:mc_halt;				//暂停功能块
	Home:mc_home;				//寻参功能块
	SetZero:mc_Setposition;		//强制设置位置功能块
	Dir: MC_Direction;			//匀速运动方向变量，1/3
	Signal:BOOL;				//寻参触发点
	temp:LREAL;
	flag:INT:=0;
	moveRelative_do: BOOL;
	temp_position: LREAL;
	temp_velocity: LREAL;
	start_position: LREAL;
	start_flag: BOOL:=TRUE;
	coefficient:INT:=1;
END_VAR

IF Axis.NcToPlc.ActPos+341.5>180 THEN
	temp:=360;
ELSIF Axis.NcToPlc.ActPos+341.5<-180	THEN
	temp:=-360;
ELSE
	temp:=0;		
END_IF
AxisOutput.Position:=Axis.NcToPlc.ActPos+341.5-temp;
IF start_flag THEN
	start_position:=AxisOutput.Position;
	start_flag:=FALSE;
END_IF
IF AxisOutput.Enable=FALSE THEN
	start_flag:=TRUE;
END_IF
AxisOutput.Velocity:=Axis.NcToPlc.ActVelo;
power(
	Axis:=axis, 
	Enable:=AxisInput.Enable, 
	Enable_Positive:=TRUE, 
	Enable_Negative:=TRUE, 
	Override:= , 
	BufferMode:= , 
	Options:= , 
	Status=>AxisOutput.Enable, 
	Busy=> , 
	Active=> , 
	Error=> , 
	ErrorID=> );
IF 	AxisOutput.Enable AND flag=0 THEN
	moveRelative_do:=TRUE;
	temp_position:=0.3;
	temp_velocity:=1;
	flag:=1;
END_IF
IF flag=1 AND AxisOutput.Position-start_position>0.2 THEN
	moveRelative_do:=AxisInput.Move_Relative;
	flag:=2;
END_IF
IF AxisOutput.Enable=FALSE AND flag=2 THEN
	flag:=0;
	moveRelative_do:=AxisInput.Move_Relative;
	temp_position:=AxisInput.Position;
	temp_velocity:=AxisInput.Velocity;
END_IF	
moveAbsolute(
	Axis:=axis, 
	Execute:=AxisInput.Move_Absolute, 
	Position:=AxisInput.Position-341.5+temp, 
	Velocity:=AxisInput.Velocity, 
	Acceleration:= , 
	Deceleration:= , 
	Jerk:= , 
	BufferMode:= , 
	Options:= , 
	Done=> , 
	Busy=> ,
	Active=> , 
	CommandAborted=> , 
	Error=> , 
	ErrorID=> );

moveRelative(
	Axis:=axis, 
	Execute:=moveRelative_do, 
	Distance:=temp_position, 
	Velocity:=temp_velocity, 
	Acceleration:= , 
	Deceleration:= , 
	Jerk:= , 
	BufferMode:= , 
	Options:= , 
	Done=> , 
	Busy=> , 
	Active=> , 
	CommandAborted=> , 
	Error=> , 
	ErrorID=> );

	IF(AxisInput.Velocity>=0)THEN
		Dir:=1;
	ELSIF(AxisInput.Velocity<0)THEN
		Dir:=3;
		AxisInput.Velocity:=-AxisInput.Velocity;
	END_IF
moveVelocity(
	Axis:= axis, 
	Execute:= AxisInput.Move_Velocity, 
	Velocity:= AxisInput.Velocity, 
	Acceleration:= , 
	Deceleration:= , 
	Jerk:= , 
	Direction:= Dir, 
	BufferMode:= , 
	Options:= , 
	InVelocity=> , 
	Busy=> , 
	Active=> , 
	CommandAborted=> , 
	Error=> , 
	ErrorID=> );
	
reset(
	Axis:= axis, 
	Execute:= AxisInput.Reset, 
	Done=> , 
	Busy=> , 
	Error=> , 
	ErrorID=> );
	
halt(
	Axis:= axis, 
	Execute:= AxisInput.Halt, 
	Deceleration:= , 
	Jerk:= , 
	BufferMode:= , 
	Options:= , 
	Done=> , 
	Busy=> , 
	Active=> , 
	CommandAborted=> , 
	Error=> , 
	ErrorID=> );
	IF(AxisInput.HomeSignal=524288)THEN
		Signal:=TRUE;
	ELSE 
		Signal:=FALSE;		
	END_IF	
Home(
	Axis:= axis, 
	Execute:= AxisInput.Home, 
	Position:=0 , 
	HomingMode:= , 
	BufferMode:= , 
	Options:= , 
	bCalibrationCam:= Signal, 
	Done=> , 
	Busy=> , 
	Active=> , 
	CommandAborted=> , 
	Error=> , 
	ErrorID=> );
	
SetZero(
	Axis:=axis , 
	Execute:=AxisInput.SetZero , 
	Position:= 0, 
	Mode:= , 
	Options:= , 
	Done=> , 
	Busy=> , 
	Error=> , 
	ErrorID=> );

END_FUNCTION_BLOCK

// ---- POUs/Rotation.TcPOU
FUNCTION_BLOCK Rotation
VAR_INPUT
	AxisInput:Command;//定义一个驱动轮PLC轴的输入结构体变量
END_VAR
VAR_OUTPUT
	AxisOutput:Status;//定义一个驱动轮PLC轴的输出结构体变量
END_VAR
VAR
	axis:axis_ref;		//定义一个轴
	power:mc_power;		//使能功能块
	moveAbsolute:mc_moveabsolute;//绝对运动功能块
	moveRelative:mc_moverelative;//相对运动功能块
	moveVelocity:mc_movevelocity;//匀速运动功能块
	reset:mc_reset;				//复位功能块
	halt:mc_halt;				//暂停功能块
	Home:mc_home;				//寻参功能块
	SetZero:mc_Setposition;		//强制设置位置功能块
	Dir: MC_Direction;			//匀速运动方向变量，1/3
	Signal:BOOL;				//寻参触发点
END_VAR

power(
	Axis:=axis, 
	Enable:=AxisInput.Enable, 
	Enable_Positive:=TRUE, 
	Enable_Negative:=TRUE, 
	Override:= , 
	BufferMode:= , 
	Options:= , 
	Status=>AxisOutput.Enable, 
	Busy=> , 
	Active=> , 
	Error=> , 
	ErrorID=> );
	
moveAbsolute(
	Axis:=axis, 
	Execute:=AxisInput.Move_Absolute, 
	Position:=AxisInput.Position+135.5, 
	Velocity:=AxisInput.Velocity, 
	Acceleration:= , 
	Deceleration:= , 
	Jerk:= , 
	BufferMode:= , 
	Options:= , 
	Done=> , 
	Busy=> , 
	Active=> , 
	CommandAborted=> , 
	Error=> , 
	ErrorID=> );

moveRelative(
	Axis:=axis, 
	Execute:=AxisInput.Move_Relative, 
	Distance:=AxisInput.Position, 
	Velocity:=AxisInput.Velocity, 
	Acceleration:= , 
	Deceleration:= , 
	Jerk:= , 
	BufferMode:= , 
	Options:= , 
	Done=> , 
	Busy=> , 
	Active=> , 
	CommandAborted=> , 
	Error=> , 
	ErrorID=> );

	IF(AxisInput.Velocity>=0)THEN
		Dir:=1;
	ELSIF(AxisInput.Velocity<0)THEN
		Dir:=3;
		AxisInput.Velocity:=-AxisInput.Velocity;
	END_IF
moveVelocity(
	Axis:= axis, 
	Execute:= AxisInput.Move_Velocity, 
	Velocity:= AxisInput.Velocity, 
	Acceleration:= , 
	Deceleration:= , 
	Jerk:= , 
	Direction:= Dir, 
	BufferMode:= , 
	Options:= , 
	InVelocity=> , 
	Busy=> , 
	Active=> , 
	CommandAborted=> , 
	Error=> , 
	ErrorID=> );
	
reset(
	Axis:= axis, 
	Execute:= AxisInput.Reset, 
	Done=> , 
	Busy=> , 
	Error=> , 
	ErrorID=> );
	
halt(
	Axis:= axis, 
	Execute:= AxisInput.Halt, 
	Deceleration:= , 
	Jerk:= , 
	BufferMode:= , 
	Options:= , 
	Done=> , 
	Busy=> , 
	Active=> , 
	CommandAborted=> , 
	Error=> , 
	ErrorID=> );
	IF(AxisInput.HomeSignal=524288)THEN
		Signal:=TRUE;
	ELSE 
		Signal:=FALSE;		
	END_IF	
Home(
	Axis:= axis, 
	Execute:= AxisInput.Home, 
	Position:= 0, 
	HomingMode:= , 
	BufferMode:= , 
	Options:= , 
	bCalibrationCam:= Signal, 
	Done=> , 
	Busy=> , 
	Active=> , 
	CommandAborted=> , 
	Error=> , 
	ErrorID=> );
	
SetZero(
	Axis:=axis , 
	Execute:=AxisInput.SetZero , 
	Position:= 0, 
	Mode:= , 
	Options:= , 
	Done=> , 
	Busy=> , 
	Error=> , 
	ErrorID=> );
AxisOutput.Position:=Axis.NcToPlc.ActPos-135.5;
AxisOutput.Velocity:=Axis.NcToPlc.ActVelo;

END_FUNCTION_BLOCK

// ---- POUs/Clamp.TcPOU
FUNCTION_BLOCK Clamp
VAR_INPUT
	AxisInput:Command;//定义一个驱动轮PLC轴的输入结构体变量
END_VAR
VAR_OUTPUT
	AxisOutput:Status;//定义一个驱动轮PLC轴的输出结构体变量
END_VAR
VAR
	axis:axis_ref;		//定义一个轴
	power:mc_power;		//使能功能块
	moveAbsolute:mc_moveabsolute;//绝对运动功能块
	moveRelative:mc_moverelative;//相对运动功能块
	moveVelocity:mc_movevelocity;//匀速运动功能块
	reset:mc_reset;				//复位功能块
	halt:mc_halt;				//暂停功能块
	Home:mc_home;				//寻参功能块
	SetZero:mc_Setposition;		//强制设置位置功能块
	Dir: MC_Direction;			//匀速运动方向变量，1/3
	Signal:BOOL;				//寻参触发点
END_VAR

power(
	Axis:=axis, 
	Enable:=AxisInput.Enable, 
	Enable_Positive:=TRUE, 
	Enable_Negative:=TRUE, 
	Override:= , 
	BufferMode:= , 
	Options:= , 
	Status=>AxisOutput.Enable, 
	Busy=> , 
	Active=> , 
	Error=> , 
	ErrorID=> );
	
moveAbsolute(
	Axis:=axis, 
	Execute:=AxisInput.Move_Absolute, 
	Position:=AxisInput.Position, 
	Velocity:=AxisInput.Velocity, 
	Acceleration:= , 
	Deceleration:= , 
	Jerk:= , 
	BufferMode:= , 
	Options:= , 
	Done=> , 
	Busy=> , 
	Active=> , 
	CommandAborted=> , 
	Error=> , 
	ErrorID=> );

moveRelative(
	Axis:=axis, 
	Execute:=AxisInput.Move_Relative, 
	Distance:=AxisInput.Position, 
	Velocity:=AxisInput.Velocity, 
	Acceleration:= , 
	Deceleration:= , 
	Jerk:= , 
	BufferMode:= , 
	Options:= , 
	Done=> , 
	Busy=> , 
	Active=> , 
	CommandAborted=> , 
	Error=> , 
	ErrorID=> );

	
	IF(AxisInput.Velocity>=0)THEN
		Dir:=1;
	ELSIF(AxisInput.Velocity<0)THEN
		Dir:=3;
		AxisInput.Velocity:=-AxisInput.Velocity;
	END_IF
moveVelocity(
	Axis:= axis, 
	Execute:= AxisInput.Move_Velocity, 
	Velocity:= AxisInput.Velocity, 
	Acceleration:= , 
	Deceleration:= , 
	Jerk:= , 
	Direction:= Dir, 
	BufferMode:= , 
	Options:= , 
	InVelocity=> , 
	Busy=> , 
	Active=> , 
	CommandAborted=> , 
	Error=> , 
	ErrorID=> );
	
reset(
	Axis:= axis, 
	Execute:= AxisInput.Reset, 
	Done=> , 
	Busy=> , 
	Error=> , 
	ErrorID=> );
	
halt(
	Axis:= axis, 
	Execute:= AxisInput.Halt, 
	Deceleration:= , 
	Jerk:= , 
	BufferMode:= , 
	Options:= , 
	Done=> , 
	Busy=> , 
	Active=> , 
	CommandAborted=> , 
	Error=> , 
	ErrorID=> );
	IF(AxisInput.HomeSignal=524288)THEN
		Signal:=TRUE;
	ELSE 
		Signal:=FALSE;		
	END_IF	
Home(
	Axis:= axis, 
	Execute:= AxisInput.Home, 
	Position:= 0, 
	HomingMode:= , 
	BufferMode:= , 
	Options:= , 
	bCalibrationCam:= Signal, 
	Done=> , 
	Busy=> , 
	Active=> , 
	CommandAborted=> , 
	Error=> , 
	ErrorID=> );
	
SetZero(
	Axis:=axis , 
	Execute:=AxisInput.SetZero , 
	Position:= 0, 
	Mode:= , 
	Options:= , 
	Done=> , 
	Busy=> , 
	Error=> , 
	ErrorID=> );
AxisOutput.Position:=Axis.NcToPlc.ActPos;
AxisOutput.Velocity:=Axis.NcToPlc.ActVelo;

END_FUNCTION_BLOCK
